C09144=1173.692,390.486,-82.941,-176.048,9.091,148.691
C09145=1173.688,390.734,-82.976,-176.048,9.094,148.691
C09146=1173.685,390.981,-83.012,-176.048,9.097,148.692
C09147=1173.681,391.228,-83.048,-176.047,9.099,148.693
C09148=1173.676,391.513,-83.089,-176.048,9.103,148.694
C09149=1173.671,391.797,-83.131,-176.047,9.107,148.694
C09150=1173.666,392.082,-83.172,-176.047,9.109,148.695
C09151=1173.663,392.366,-83.213,-176.047,9.112,148.696
C09152=1173.658,392.614,-83.249,-176.047,9.115,148.697
C09153=1173.654,392.861,-83.285,-176.047,9.118,148.697
C09154=1173.651,393.109,-83.320,-176.047,9.121,148.698
C09155=1173.647,393.356,-83.356,-176.047,9.124,148.699
C09156=1173.643,393.604,-83.392,-176.047,9.126,148.699
C09157=1173.639,393.851,-83.428,-176.047,9.129,148.700
C09158=1173.636,394.099,-83.464,-176.046,9.132,148.701
C09159=1173.631,394.346,-83.499,-176.047,9.134,148.701
C09160=1173.627,394.593,-83.535,-176.047,9.137,148.702
C09161=1173.623,394.841,-83.570,-176.047,9.140,148.703
C09162=1173.619,395.088,-83.607,-176.047,9.142,148.704
C09163=1173.616,395.335,-83.643,-176.047,9.145,148.704
C09164=1173.611,395.583,-83.679,-176.047,9.147,148.705
C09165=1173.608,395.831,-83.715,-176.047,9.150,148.706
C09166=1173.604,396.078,-83.751,-176.047,9.152,148.706
C09167=1173.599,396.325,-83.787,-176.047,9.155,148.707
C09168=1173.596,396.572,-83.822,-176.048,9.157,148.708
C09169=1173.592,396.820,-83.858,-176.048,9.160,148.708
C09170=1173.588,397.067,-83.895,-176.048,9.162,148.709
C09171=1173.584,397.314,-83.930,-176.048,9.165,148.710
C09172=1173.580,397.562,-83.966,-176.048,9.167,148.711
C09173=1173.576,397.810,-84.002,-176.048,9.170,148.711
C09174=1173.573,398.057,-84.038,-176.048,9.172,148.712
C09175=1173.568,398.304,-84.074,-176.048,9.175,148.713
C09176=1173.564,398.551,-84.109,-176.048,9.177,148.713
C09177=1173.561,398.798,-84.146,-176.049,9.180,148.714
C09178=1173.556,399.046,-84.182,-176.049,9.183,148.715
C09179=1173.553,399.293,-84.217,-176.049,9.185,148.715
C09180=1173.548,399.541,-84.253,-176.049,9.187,148.716
C09181=1173.545,399.788,-84.290,-176.049,9.189,148.717
C09182=1173.541,400.036,-84.325,-176.049,9.192,148.717
C09183=1173.537,400.283,-84.361,-176.050,9.194,148.718
C09184=1173.533,400.530,-84.398,-176.050,9.197,148.719
C09185=1173.529,400.778,-84.434,-176.050,9.198,148.719
C09186=1173.525,401.026,-84.469,-176.050,9.201,148.720
C09187=1173.521,401.272,-84.505,-176.050,9.203,148.721
C09188=1173.517,401.520,-84.541,-176.050,9.206,148.721
C09189=1173.513,401.767,-84.577,-176.051,9.208,148.722
C09190=1173.509,402.014,-84.614,-176.051,9.210,148.722
C09191=1173.506,402.262,-84.649,-176.051,9.213,148.723
C09192=1173.501,402.510,-84.686,-176.052,9.214,148.724
C09193=1173.498,402.757,-84.722,-176.052,9.217,148.725
C09194=1173.494,403.004,-84.757,-176.052,9.219,148.725
C09195=1173.490,403.252,-84.793,-176.052,9.221,148.726
C09196=1173.486,403.499,-84.830,-176.053,9.223,148.726
C09197=1173.482,403.747,-84.866,-176.052,9.226,148.727
C09198=1173.479,403.993,-84.902,-176.053,9.227,148.728
C09199=1173.474,404.240,-84.938,-176.053,9.230,148.728
C09200=1173.470,404.488,-84.973,-176.053,9.233,148.729
C09201=1173.467,404.735,-85.010,-176.054,9.234,148.729
C09202=1173.462,404.983,-85.046,-176.054,9.237,148.730
C09203=1173.459,405.230,-85.081,-176.054,9.238,148.731
C09204=1173.455,405.477,-85.118,-176.054,9.241,148.731
C09205=1173.451,405.725,-85.154,-176.055,9.242,148.732
C09206=1173.447,405.972,-85.191,-176.055,9.245,148.733
C09207=1173.443,406.220,-85.226,-176.055,9.246,148.733
C09208=1173.439,406.467,-85.262,-176.056,9.249,148.734
C09209=1173.435,406.714,-85.299,-176.055,9.251,148.734
C09210=1173.432,406.962,-85.334,-176.056,9.253,148.735
C09211=1173.428,407.209,-85.371,-176.056,9.255,148.736
C09212=1173.424,407.456,-85.407,-176.056,9.257,148.736
C09213=1173.420,407.704,-85.443,-176.057,9.259,148.737
C09214=1173.416,407.951,-85.479,-176.057,9.261,148.737
C09215=1173.412,408.199,-85.515,-176.057,9.263,148.738
C09216=1173.408,408.445,-85.551,-176.058,9.265,148.739
C09217=1173.403,408.693,-85.587,-176.058,9.267,148.739
C09218=1173.400,408.940,-85.623,-176.058,9.269,148.740
C09219=1173.396,409.188,-85.660,-176.058,9.271,148.740
C09220=1173.392,409.435,-85.695,-176.059,9.273,148.741
C09221=1173.388,409.682,-85.732,-176.059,9.275,148.742
C09222=1173.384,409.930,-85.768,-176.059,9.277,148.742
C09223=1173.381,410.177,-85.804,-176.059,9.279,148.743
C09224=1173.376,410.425,-85.840,-176.059,9.281,148.743
C09225=1173.373,410.672,-85.875,-176.060,9.283,148.744
C09226=1173.369,410.919,-85.912,-176.060,9.284,148.745
C09227=1173.365,411.167,-85.948,-176.060,9.287,148.745
C09228=1173.361,411.414,-85.985,-176.061,9.288,148.746
C09229=1173.357,411.661,-86.020,-176.061,9.291,148.746
C09230=1173.353,411.909,-86.057,-176.061,9.292,148.747
C09231=1173.350,412.156,-86.093,-176.062,9.294,148.747
C09232=1173.345,412.403,-86.130,-176.061,9.296,148.748
C09233=1173.342,412.651,-86.165,-176.062,9.298,148.749
C09234=1173.338,412.898,-86.202,-176.062,9.300,148.749
C09235=1173.334,413.145,-86.238,-176.062,9.302,148.750
C09236=1173.330,413.393,-86.274,-176.063,9.303,148.750
C09237=1173.326,413.640,-86.310,-176.063,9.306,148.751
C09238=1173.322,413.887,-86.347,-176.063,9.307,148.751
C09239=1173.318,414.135,-86.382,-176.064,9.309,148.752
C09240=1173.314,414.383,-86.418,-176.063,9.311,148.752
C09241=1173.310,414.629,-86.454,-176.064,9.313,148.753
C09242=1173.306,414.877,-86.491,-176.064,9.314,148.753
C09243=1173.302,415.124,-86.527,-176.064,9.316,148.754
C09244=1173.298,415.371,-86.563,-176.065,9.318,148.755
C09245=1173.295,415.619,-86.600,-176.065,9.320,148.755
C09246=1173.292,415.866,-86.636,-176.065,9.322,148.756
C09247=1173.291,416.113,-86.672,-176.065,9.323,148.756
C09248=1173.290,416.376,-86.709,-176.065,9.325,148.756
C09249=1173.291,416.639,-86.748,-176.065,9.327,148.757
C09250=1173.293,416.901,-86.785,-176.066,9.329,148.758
C09251=1173.296,417.163,-86.823,-176.066,9.330,148.758
C09252=1172.876,417.164,-86.867,-176.069,9.341,148.762
C09253=1172.873,416.899,-86.829,-176.069,9.339,148.761
C09254=1172.871,416.634,-86.790,-176.068,9.338,148.761
C09255=1172.869,416.368,-86.752,-176.069,9.336,148.760
C09256=1172.870,416.102,-86.714,-176.068,9.334,148.760
C09257=1172.872,415.855,-86.678,-176.068,9.333,148.759
C09258=1172.874,415.607,-86.642,-176.068,9.330,148.759
C09259=1172.877,415.361,-86.606,-176.068,9.329,148.758
C09260=1172.882,415.113,-86.570,-176.067,9.327,148.758
C09261=1172.885,414.866,-86.533,-176.067,9.325,148.757
C09262=1172.889,414.618,-86.497,-176.067,9.323,148.757
C09263=1172.893,414.371,-86.461,-176.067,9.322,148.756
C09264=1172.897,414.123,-86.425,-176.066,9.319,148.755
C09265=1172.901,413.876,-86.389,-176.066,9.318,148.755
C09266=1172.905,413.629,-86.352,-176.066,9.317,148.754
C09267=1172.908,413.382,-86.316,-176.066,9.314,148.754
C09268=1172.913,413.134,-86.280,-176.065,9.313,148.753
C09269=1172.916,412.887,-86.244,-176.065,9.311,148.753
C09270=1172.921,412.639,-86.208,-176.065,9.309,148.752
C09271=1172.924,412.392,-86.171,-176.065,9.307,148.752
C09272=1172.928,412.145,-86.135,-176.065,9.305,148.751
C09273=1172.932,411.898,-86.099,-176.064,9.303,148.751
C09274=1172.936,411.650,-86.063,-176.064,9.301,148.750
C09275=1172.939,411.403,-86.026,-176.064,9.299,148.749
C09276=1172.944,411.155,-85.990,-176.063,9.297,148.749
C09277=1172.947,410.908,-85.954,-176.063,9.296,148.748
C09278=1172.952,410.661,-85.918,-176.063,9.293,148.748
C09279=1172.955,410.413,-85.882,-176.062,9.292,148.747
C09280=1172.959,410.166,-85.846,-176.062,9.289,148.746
C09281=1172.963,409.918,-85.810,-176.062,9.288,148.746
C09282=1172.967,409.671,-85.773,-176.062,9.285,148.745
C09283=1172.971,409.424,-85.738,-176.061,9.284,148.745
C09284=1172.975,409.176,-85.701,-176.061,9.282,148.744
C09285=1172.978,408.929,-85.665,-176.061,9.280,148.744
C09286=1172.983,408.682,-85.629,-176.060,9.278,148.743
C09287=1172.987,408.435,-85.593,-176.061,9.276,148.742
C09288=1172.991,408.187,-85.557,-176.060,9.274,148.742
C09289=1172.995,407.940,-85.521,-176.060,9.272,148.741
C09290=1172.999,407.692,-85.485,-176.059,9.270,148.741
C09291=1173.002,407.446,-85.448,-176.059,9.268,148.740
C09292=1173.006,407.198,-85.413,-176.059,9.266,148.739
C09293=1173.010,406.951,-85.376,-176.059,9.264,148.739
C09294=1173.014,406.703,-85.340,-176.059,9.262,148.738
C09295=1173.018,406.456,-85.304,-176.058,9.260,148.738
C09296=1173.022,406.209,-85.268,-176.058,9.258,148.737
C09297=1173.026,405.961,-85.232,-176.058,9.256,148.736
C09298=1173.029,405.714,-85.196,-176.057,9.254,148.736
C09299=1173.034,405.466,-85.159,-176.057,9.251,148.735
C09300=1173.037,405.219,-85.124,-176.057,9.250,148.735
C09301=1173.041,404.971,-85.087,-176.057,9.247,148.734
C09302=1173.045,404.724,-85.051,-176.056,9.246,148.733
C09303=1173.048,404.477,-85.015,-176.056,9.243,148.733
C09304=1173.053,404.230,-84.979,-176.056,9.241,148.732
C09305=1173.057,403.983,-84.944,-176.055,9.239,148.731
C09306=1173.061,403.735,-84.907,-176.055,9.236,148.731
C09307=1173.065,403.488,-84.871,-176.055,9.235,148.730
C09308=1173.069,403.240,-84.835,-176.055,9.232,148.729
C09309=1173.073,402.993,-84.799,-176.055,9.230,148.729
C09310=1173.077,402.745,-84.763,-176.054,9.228,148.728
C09311=1173.081,402.498,-84.727,-176.054,9.226,148.727
C09312=1173.084,402.251,-84.691,-176.054,9.223,148.727
C09313=1173.088,402.003,-84.655,-176.053,9.221,148.726
C09314=1173.092,401.756,-84.619,-176.053,9.219,148.725
C09315=1173.096,401.508,-84.583,-176.053,9.217,148.725
C09316=1173.100,401.261,-84.547,-176.053,9.214,148.724
C09317=1173.103,401.014,-84.511,-176.053,9.212,148.724
C09318=1173.108,400.767,-84.475,-176.052,9.210,148.723
C09319=1173.112,400.519,-84.439,-176.052,9.207,148.722
C09320=1173.116,400.272,-84.403,-176.052,9.205,148.721
C09321=1173.120,400.025,-84.367,-176.052,9.203,148.721
C09322=1173.124,399.777,-84.331,-176.052,9.201,148.720
C09323=1173.127,399.530,-84.295,-176.051,9.198,148.719
C09324=1173.131,399.283,-84.259,-176.051,9.195,148.719
C09325=1173.135,399.035,-84.223,-176.051,9.193,148.718
C09326=1173.139,398.787,-84.187,-176.050,9.191,148.717
C09327=1173.143,398.540,-84.151,-176.051,9.189,148.717
C09328=1173.147,398.293,-84.115,-176.051,9.186,148.716
C09329=1173.151,398.046,-84.080,-176.050,9.184,148.715
C09330=1173.155,397.799,-84.043,-176.050,9.181,148.715
C09331=1173.159,397.551,-84.007,-176.050,9.179,148.714
C09332=1173.163,397.303,-83.971,-176.050,9.176,148.713
C09333=1173.167,397.056,-83.936,-176.050,9.174,148.713
C09334=1173.170,396.809,-83.899,-176.050,9.171,148.712
C09335=1173.175,396.561,-83.863,-176.050,9.169,148.711
C09336=1173.178,396.314,-83.828,-176.050,9.166,148.711
C09337=1173.182,396.067,-83.791,-176.050,9.164,148.710
C09338=1173.187,395.820,-83.756,-176.049,9.161,148.709
C09339=1173.190,395.572,-83.720,-176.049,9.158,148.708
C09340=1173.195,395.324,-83.684,-176.049,9.156,148.708
C09341=1173.198,395.077,-83.648,-176.049,9.153,148.707
C09342=1173.202,394.830,-83.612,-176.049,9.151,148.706
C09343=1173.206,394.582,-83.576,-176.049,9.148,148.706
C09344=1173.210,394.335,-83.541,-176.049,9.146,148.705
C09345=1173.214,394.087,-83.505,-176.049,9.142,148.704
C09346=1173.218,393.840,-83.468,-176.049,9.140,148.704
C09347=1173.222,393.593,-83.433,-176.049,9.137,148.703
C09348=1173.226,393.346,-83.397,-176.049,9.135,148.702
C09349=1173.230,393.098,-83.361,-176.049,9.132,148.701
C09350=1173.233,392.851,-83.325,-176.049,9.129,148.701
C09351=1173.237,392.603,-83.289,-176.049,9.126,148.700
C09352=1173.241,392.356,-83.253,-176.049,9.124,148.699
C09353=1173.246,392.071,-83.213,-176.049,9.120,148.698
C09354=1173.250,391.786,-83.171,-176.049,9.118,148.698
C09355=1173.255,391.501,-83.130,-176.049,9.114,148.697
C09356=1173.259,391.217,-83.089,-176.049,9.111,148.696
C09357=1173.263,390.970,-83.053,-176.050,9.108,148.696
C09358=1173.267,390.722,-83.017,-176.050,9.105,148.695
C09359=1173.271,390.475,-82.982,-176.050,9.102,148.694
C09360=1173.276,390.227,-82.946,-176.050,9.099,148.693
C09361=1173.279,389.981,-82.910,-176.050,9.096,148.693
C09362=1173.283,389.733,-82.874,-176.051,9.093,148.692
C09363=1173.286,389.486,-82.839,-176.051,9.091,148.691
C09364=1173.291,389.238,-82.802,-176.051,9.087,148.690
C09365=1173.295,388.991,-82.767,-176.051,9.085,148.690
C09366=1173.299,388.743,-82.732,-176.052,9.081,148.689
C09367=1173.302,388.496,-82.696,-176.052,9.078,148.688
C09368=1173.307,388.248,-82.660,-176.052,9.076,148.688
C09369=1173.310,388.001,-82.624,-176.053,9.072,148.687
C09370=1173.314,387.754,-82.588,-176.052,9.070,148.686
C09371=1173.319,387.507,-82.552,-176.053,9.067,148.686
C09372=1173.322,387.259,-82.517,-176.054,9.063,148.685
C09373=1173.326,387.012,-82.481,-176.054,9.060,148.684
C09374=1173.330,386.764,-82.446,-176.054,9.058,148.684
C09375=1173.333,386.517,-82.410,-176.055,9.054,148.683
C09376=1173.338,386.269,-82.374,-176.055,9.051,148.682
C09377=1173.342,386.022,-82.339,-176.056,9.048,148.681
C09378=1173.346,385.775,-82.303,-176.056,9.044,148.681
C09379=1173.349,385.527,-82.268,-176.057,9.041,148.680
C09380=1173.354,385.279,-82.232,-176.058,9.038,148.679
C09381=1173.357,385.032,-82.196,-176.058,9.035,148.679
C09382=1173.362,384.785,-82.161,-176.059,9.031,148.678
C09383=1173.365,384.537,-82.125,-176.059,9.028,148.677
C09384=1173.369,384.290,-82.090,-176.060,9.025,148.677
C09385=1173.373,384.042,-82.054,-176.061,9.022,148.676
C09386=1173.377,383.795,-82.018,-176.061,9.018,148.675
C09387=1173.381,383.548,-81.983,-176.062,9.015,148.674
C09388=1173.385,383.300,-81.947,-176.063,9.012,148.674
C09389=1173.389,383.053,-81.912,-176.064,9.009,148.673
C09390=1173.392,382.805,-81.876,-176.064,9.006,148.673
C09391=1173.398,382.558,-81.841,-176.065,9.002,148.672
C09392=1173.401,382.310,-81.806,-176.066,8.998,148.671
C09393=1173.405,382.063,-81.770,-176.067,8.995,148.671
C09394=1173.409,381.815,-81.735,-176.067,8.992,148.670
C09395=1173.413,381.568,-81.699,-176.068,8.989,148.669
C09396=1173.416,381.321,-81.664,-176.069,8.986,148.669
C09397=1173.420,381.073,-81.628,-176.070,8.982,148.668
C09398=1173.425,380.825,-81.592,-176.071,8.979,148.667
C09399=1173.429,380.578,-81.558,-176.071,8.975,148.667
C09400=1173.433,380.331,-81.522,-176.073,8.971,148.666
C09401=1173.436,380.083,-81.487,-176.074,8.968,148.665
C09402=1173.440,379.836,-81.451,-176.074,8.965,148.665
C09403=1173.444,379.589,-81.416,-176.076,8.961,148.664
C09404=1173.448,379.341,-81.380,-176.077,8.958,148.664
C09405=1173.452,379.093,-81.345,-176.078,8.954,148.663
C09406=1173.456,378.846,-81.310,-176.079,8.951,148.662
C09407=1173.460,378.599,-81.275,-176.080,8.947,148.662
C09408=1173.464,378.351,-81.239,-176.081,8.944,148.661
C09409=1173.468,378.103,-81.204,-176.082,8.940,148.660
C09410=1173.473,377.856,-81.169,-176.083,8.937,148.660
C09411=1173.476,377.609,-81.133,-176.084,8.933,148.659
C09412=1173.480,377.361,-81.098,-176.086,8.930,148.659
C09413=1173.484,377.114,-81.063,-176.087,8.926,148.658
C09414=1173.488,376.866,-81.028,-176.088,8.923,148.658
C09415=1173.492,376.619,-80.992,-176.089,8.919,148.657
C09416=1173.496,376.371,-80.957,-176.091,8.915,148.656
C09417=1173.500,376.124,-80.922,-176.092,8.912,148.656
C09418=1173.504,375.876,-80.886,-176.093,8.908,148.655
C09419=1173.508,375.628,-80.852,-176.095,8.905,148.655
C09420=1173.512,375.381,-80.816,-176.096,8.902,148.654
C09421=1173.516,375.134,-80.781,-176.097,8.898,148.653
C09422=1173.519,374.886,-80.746,-176.098,8.894,148.653
C09423=1173.524,374.639,-80.711,-176.100,8.891,148.652
C09424=1173.527,374.391,-80.675,-176.101,8.887,148.652
C09425=1173.531,374.144,-80.641,-176.103,8.883,148.651
C09426=1173.535,373.897,-80.606,-176.104,8.879,148.651
C09427=1173.539,373.649,-80.571,-176.105,8.876,148.650
C09428=1173.543,373.402,-80.536,-176.107,8.872,148.650
C09429=1173.547,373.154,-80.501,-176.108,8.869,148.649
C09430=1173.551,372.906,-80.465,-176.110,8.865,148.649
C09431=1173.555,372.659,-80.431,-176.112,8.861,148.648
C09432=1173.559,372.411,-80.395,-176.113,8.857,148.647
C09433=1173.563,372.163,-80.361,-176.114,8.855,148.647
C09434=1173.567,371.916,-80.325,-176.116,8.851,148.646
C09435=1173.571,371.668,-80.291,-176.118,8.847,148.646
C09436=1173.575,371.422,-80.256,-176.119,8.843,148.646
C09437=1173.579,371.174,-80.221,-176.121,8.840,148.645
C09438=1173.582,370.926,-80.186,-176.123,8.836,148.645
C09439=1173.587,370.679,-80.151,-176.125,8.832,148.644
C09440=1173.591,370.431,-80.116,-176.126,8.828,148.643
C09441=1173.595,370.184,-80.081,-176.128,8.825,148.643
C09442=1173.599,369.936,-80.046,-176.130,8.821,148.643
C09443=1173.603,369.689,-80.012,-176.131,8.817,148.642
C09444=1173.607,369.441,-79.977,-176.133,8.814,148.642
C09445=1173.611,369.193,-79.942,-176.135,8.810,148.641
C09446=1173.615,368.946,-79.907,-176.137,8.806,148.641
C09447=1173.619,368.698,-79.872,-176.138,8.803,148.640
C09448=1173.623,368.451,-79.838,-176.140,8.799,148.640
C09449=1173.626,368.203,-79.803,-176.142,8.795,148.639
C09450=1173.631,367.956,-79.768,-176.143,8.792,148.639
C09451=1173.635,367.708,-79.733,-176.145,8.788,148.638
C09452=1173.638,367.461,-79.699,-176.147,8.785,148.638
C09453=1173.642,367.213,-79.664,-176.149,8.781,148.637
C09454=1173.647,366.966,-79.629,-176.151,8.777,148.637
C09455=1173.651,366.718,-79.595,-176.153,8.774,148.637
C09456=1173.655,366.471,-79.561,-176.154,8.770,148.636
C09457=1173.659,366.188,-79.521,-176.157,8.766,148.636
C09458=1173.664,365.907,-79.481,-176.159,8.762,148.635
C09459=1173.668,365.624,-79.442,-176.161,8.758,148.635
C09460=1173.673,365.343,-79.402,-176.164,8.753,148.634
C09461=1173.676,365.095,-79.368,-176.165,8.750,148.634
C09462=1173.681,364.847,-79.333,-176.167,8.746,148.633
C09463=1173.685,364.599,-79.299,-176.169,8.743,148.633
C09464=1173.688,364.353,-79.264,-176.171,8.739,148.633
C09465=1173.692,364.105,-79.229,-176.174,8.735,148.632
C09466=1173.697,363.857,-79.195,-176.176,8.731,148.632
C09467=1173.701,363.610,-79.161,-176.178,8.728,148.632
C09468=1173.705,363.362,-79.126,-176.180,8.724,148.631
C09469=1173.709,363.115,-79.092,-176.182,8.720,148.631
C09470=1173.712,362.867,-79.057,-176.184,8.717,148.631
C09471=1173.717,362.619,-79.023,-176.186,8.713,148.630
C09472=1173.720,362.372,-78.989,-176.188,8.709,148.630
C09473=1173.725,362.124,-78.954,-176.190,8.706,148.629
C09474=1173.728,361.876,-78.920,-176.192,8.702,148.629
C09475=1173.733,361.629,-78.885,-176.194,8.699,148.629
C09476=1173.736,361.382,-78.852,-176.197,8.694,148.628
C09477=1173.740,361.134,-78.817,-176.199,8.691,148.628
C09478=1173.745,360.886,-78.782,-176.201,8.688,148.628
C09479=1173.748,360.639,-78.748,-176.203,8.684,148.627
C09480=1173.753,360.391,-78.714,-176.205,8.681,148.627
C09481=1173.757,360.143,-78.680,-176.207,8.676,148.627
C09482=1173.761,359.895,-78.646,-176.210,8.673,148.626
C09483=1173.765,359.648,-78.612,-176.212,8.669,148.626
C09484=1173.769,359.400,-78.577,-176.214,8.666,148.626
C09485=1173.773,359.153,-78.543,-176.216,8.662,148.625
C09486=1173.777,358.905,-78.509,-176.219,8.658,148.625
C09487=1173.781,358.657,-78.475,-176.221,8.655,148.625
C09488=1173.785,358.410,-78.441,-176.223,8.651,148.624
C09489=1173.789,358.163,-78.407,-176.225,8.648,148.624
C09490=1173.792,357.915,-78.372,-176.227,8.644,148.624
C09491=1173.797,357.667,-78.338,-176.230,8.640,148.623
C09492=1173.801,357.420,-78.305,-176.232,8.637,148.623
C09493=1173.805,357.171,-78.270,-176.234,8.633,148.623
C09494=1173.809,356.924,-78.236,-176.236,8.630,148.623
C09495=1173.813,356.677,-78.203,-176.239,8.626,148.622
C09496=1173.817,356.428,-78.168,-176.241,8.622,148.622
C09497=1173.821,356.181,-78.134,-176.243,8.619,148.622
C09498=1173.826,355.933,-78.101,-176.245,8.616,148.621
C09499=1173.829,355.686,-78.066,-176.248,8.611,148.621
C09500=1173.833,355.438,-78.032,-176.250,8.608,148.621
C09501=1173.838,355.190,-77.999,-176.252,8.605,148.621
C09502=1173.841,354.943,-77.964,-176.255,8.601,148.620
C09503=1173.845,354.695,-77.931,-176.256,8.598,148.620
C09504=1173.850,354.447,-77.897,-176.259,8.594,148.620
C09505=1173.853,354.200,-77.863,-176.261,8.590,148.619
C09506=1173.857,353.952,-77.829,-176.264,8.587,148.619
C09507=1173.861,353.704,-77.795,-176.266,8.583,148.619
C09508=1173.866,353.457,-77.762,-176.268,8.580,148.619
C09509=1173.869,353.210,-77.728,-176.271,8.576,148.618
C09510=1173.873,352.961,-77.694,-176.273,8.573,148.618
C09511=1173.878,352.714,-77.660,-176.275,8.569,148.618
C09512=1173.882,352.466,-77.627,-176.277,8.566,148.617
C09513=1173.885,352.219,-77.593,-176.279,8.562,148.617
C09514=1173.889,351.970,-77.559,-176.282,8.558,148.617
C09515=1173.894,351.723,-77.525,-176.285,8.555,148.617
C09516=1173.898,351.475,-77.492,-176.287,8.552,148.616
C09517=1173.902,351.228,-77.459,-176.289,8.548,148.616
C09518=1173.906,350.981,-77.425,-176.291,8.545,148.616
C09519=1173.910,350.732,-77.391,-176.294,8.541,148.616
C09520=1173.914,350.484,-77.357,-176.296,8.537,148.615
C09521=1173.918,350.237,-77.324,-176.298,8.534,148.615
C09522=1173.922,349.989,-77.290,-176.301,8.531,148.615
C09523=1173.926,349.741,-77.257,-176.303,8.527,148.615
C09524=1173.930,349.494,-77.223,-176.306,8.523,148.614
C09525=1173.934,349.246,-77.189,-176.308,8.520,148.614
C09526=1173.938,348.998,-77.156,-176.310,8.516,148.614
C09527=1173.942,348.751,-77.122,-176.312,8.513,148.614
C09528=1173.946,348.503,-77.089,-176.314,8.510,148.613
C09529=1173.951,348.255,-77.056,-176.317,8.506,148.613
C09530=1173.955,348.008,-77.023,-176.319,8.502,148.613
C09531=1173.959,347.760,-76.989,-176.322,8.499,148.613
C09532=1173.963,347.512,-76.955,-176.324,8.496,148.612
C09533=1173.967,347.264,-76.922,-176.326,8.492,148.612
C09534=1173.971,347.016,-76.889,-176.329,8.489,148.612
C09535=1173.975,346.769,-76.855,-176.331,8.486,148.612
C09536=1173.979,346.521,-76.822,-176.334,8.482,148.612
C09537=1173.984,346.273,-76.789,-176.336,8.478,148.611
C09538=1173.987,346.026,-76.755,-176.338,8.475,148.611
C09539=1173.991,345.778,-76.722,-176.341,8.472,148.611
C09540=1173.996,345.531,-76.689,-176.343,8.468,148.611
C09541=1174.000,345.283,-76.656,-176.345,8.465,148.610
C09542=1174.003,345.034,-76.622,-176.347,8.462,148.610
C09543=1174.007,344.787,-76.589,-176.350,8.458,148.610
C09544=1174.012,344.539,-76.556,-176.352,8.454,148.610
C09545=1174.016,344.291,-76.523,-176.355,8.451,148.610
C09546=1174.020,344.043,-76.490,-176.357,8.448,148.609
C09547=1174.024,343.796,-76.456,-176.359,8.445,148.609
C09548=1174.028,343.548,-76.423,-176.362,8.441,148.609
C09549=1174.032,343.300,-76.390,-176.364,8.438,148.609
C09550=1174.036,343.053,-76.357,-176.367,8.434,148.608
C09551=1174.041,342.805,-76.324,-176.369,8.430,148.608
C09552=1174.045,342.557,-76.291,-176.371,8.427,148.608
C09553=1174.049,342.309,-76.257,-176.374,8.424,148.608
C09554=1174.053,342.062,-76.224,-176.376,8.421,148.608
C09555=1174.057,341.813,-76.192,-176.379,8.418,148.608
C09556=1174.061,341.566,-76.159,-176.381,8.414,148.607
C09557=1174.065,341.318,-76.126,-176.384,8.410,148.607
C09558=1174.069,341.070,-76.093,-176.386,8.407,148.607
C09559=1174.073,340.823,-76.060,-176.388,8.404,148.607
C09560=1174.077,340.575,-76.027,-176.391,8.400,148.606
C09561=1174.082,340.295,-75.989,-176.393,8.396,148.606
C09562=1174.087,340.016,-75.953,-176.396,8.393,148.606
C09563=1174.091,339.737,-75.916,-176.399,8.389,148.606
C09564=1174.097,339.458,-75.879,-176.402,8.385,148.606
C09565=1174.100,339.210,-75.846,-176.404,8.382,148.605
C09566=1174.104,338.963,-75.813,-176.406,8.378,148.605
C09567=1174.108,338.714,-75.780,-176.409,8.375,148.605
C09568=1174.113,338.466,-75.747,-176.411,8.372,148.605
C09569=1174.117,338.219,-75.714,-176.414,8.369,148.605
C09570=1174.120,337.971,-75.682,-176.416,8.365,148.605
C09571=1174.125,337.723,-75.649,-176.418,8.362,148.604
C09572=1174.129,337.475,-75.616,-176.420,8.359,148.604
C09573=1174.133,337.227,-75.584,-176.423,8.355,148.604
C09574=1174.137,336.979,-75.551,-176.426,8.352,148.604
C09575=1174.141,336.732,-75.518,-176.428,8.348,148.604
C09576=1174.146,336.484,-75.486,-176.431,8.345,148.604
C09577=1174.149,336.237,-75.453,-176.433,8.342,148.603
C09578=1174.154,335.988,-75.421,-176.435,8.338,148.603
C09579=1174.158,335.741,-75.388,-176.438,8.335,148.603
C09580=1174.161,335.493,-75.356,-176.440,8.332,148.603
C09581=1174.166,335.245,-75.323,-176.442,8.329,148.603
C09582=1174.170,334.996,-75.290,-176.445,8.325,148.603
C09583=1174.173,334.749,-75.258,-176.448,8.322,148.602
C09584=1174.178,334.501,-75.225,-176.450,8.318,148.602
C09585=1174.183,334.254,-75.192,-176.452,8.315,148.602
C09586=1174.186,334.006,-75.161,-176.455,8.312,148.602
C09587=1174.190,333.758,-75.127,-176.457,8.309,148.602
C09588=1174.195,333.510,-75.095,-176.460,8.305,148.602
C09589=1174.198,333.262,-75.062,-176.462,8.302,148.601
C09590=1174.203,333.014,-75.030,-176.464,8.299,148.601
C09591=1174.207,332.767,-74.998,-176.467,8.296,148.601
C09592=1174.211,332.519,-74.965,-176.469,8.293,148.601
C09593=1174.216,332.270,-74.933,-176.472,8.289,148.601
C09594=1174.219,332.023,-74.900,-176.475,8.285,148.601
C09595=1174.224,331.775,-74.868,-176.477,8.282,148.601
C09596=1174.228,331.527,-74.836,-176.479,8.279,148.600
C09597=1174.232,331.280,-74.803,-176.482,8.276,148.600
C09598=1174.236,331.032,-74.771,-176.484,8.273,148.600
C09599=1174.240,330.783,-74.739,-176.487,8.269,148.600
C09600=1174.244,330.535,-74.707,-176.489,8.266,148.600
C09601=1174.249,330.288,-74.674,-176.492,8.263,148.600
C09602=1174.252,330.040,-74.642,-176.494,8.260,148.600
C09603=1174.257,329.792,-74.610,-176.496,8.256,148.599
C09604=1174.260,329.544,-74.578,-176.499,8.253,148.599
C09605=1174.265,329.297,-74.545,-176.501,8.250,148.599
C09606=1174.269,329.049,-74.514,-176.504,8.247,148.599
C09607=1174.273,328.800,-74.481,-176.507,8.243,148.599
C09608=1174.277,328.552,-74.449,-176.509,8.240,148.599
C09609=1174.282,328.305,-74.417,-176.512,8.237,148.599
C09610=1174.286,328.057,-74.385,-176.514,8.233,148.598
C09611=1174.290,327.809,-74.352,-176.516,8.230,148.598
C09612=1174.294,327.561,-74.320,-176.519,8.227,148.598
C09613=1174.298,327.313,-74.289,-176.521,8.224,148.598
C09614=1174.302,327.065,-74.256,-176.524,8.220,148.598
C09615=1174.306,326.817,-74.225,-176.526,8.217,148.598
C09616=1174.310,326.570,-74.193,-176.529,8.214,148.598
C09617=1174.315,326.321,-74.161,-176.531,8.211,148.598
C09618=1174.319,326.073,-74.129,-176.534,8.208,148.597
C09619=1174.324,325.826,-74.097,-176.536,8.205,148.597
C09620=1174.327,325.578,-74.065,-176.539,8.202,148.597
C09621=1174.331,325.330,-74.033,-176.541,8.198,148.597
C09622=1174.335,325.081,-74.001,-176.544,8.195,148.597
C09623=1174.340,324.834,-73.969,-176.546,8.192,148.597
C09624=1174.343,324.586,-73.937,-176.549,8.189,148.597
C09625=1174.347,324.338,-73.905,-176.551,8.186,148.597
C09626=1174.352,324.090,-73.873,-176.554,8.182,148.596
C09627=1174.356,323.842,-73.842,-176.557,8.179,148.596
C09628=1174.360,323.595,-73.810,-176.559,8.175,148.596
C09629=1174.365,323.346,-73.778,-176.562,8.172,148.596
C09630=1174.369,323.098,-73.746,-176.564,8.169,148.596
C09631=1174.373,322.850,-73.715,-176.567,8.166,148.596
C09632=1174.377,322.602,-73.683,-176.569,8.163,148.596
C09633=1174.380,322.354,-73.651,-176.571,8.159,148.596
C09634=1174.385,322.107,-73.619,-176.574,8.156,148.596
C09635=1174.389,321.859,-73.587,-176.576,8.153,148.595
C09636=1174.394,321.611,-73.557,-176.579,8.150,148.595
C09637=1174.397,321.363,-73.525,-176.581,8.147,148.595
C09638=1174.401,321.115,-73.493,-176.584,8.144,148.595
C09639=1174.406,320.867,-73.461,-176.586,8.140,148.595
C09640=1174.410,320.618,-73.430,-176.589,8.137,148.595
C09641=1174.415,320.371,-73.398,-176.591,8.134,148.595
C09642=1174.418,320.123,-73.366,-176.594,8.131,148.595
C09643=1174.422,319.875,-73.335,-176.596,8.128,148.595
C09644=1174.427,319.627,-73.304,-176.599,8.125,148.595
C09645=1174.431,319.379,-73.271,-176.601,8.122,148.595
C09646=1174.435,319.131,-73.240,-176.604,8.119,148.595
C09647=1174.439,318.883,-73.209,-176.606,8.115,148.594
C09648=1174.444,318.635,-73.177,-176.609,8.112,148.594
C09649=1174.448,318.387,-73.146,-176.611,8.109,148.594
C09650=1174.452,318.139,-73.115,-176.614,8.106,148.594
C09651=1174.456,317.891,-73.083,-176.616,8.103,148.594
C09652=1174.460,317.643,-73.052,-176.619,8.100,148.594
C09653=1174.464,317.395,-73.020,-176.621,8.096,148.594
C09654=1174.469,317.147,-72.989,-176.624,8.093,148.594
C09655=1174.472,316.899,-72.958,-176.626,8.090,148.594
C09656=1174.477,316.651,-72.927,-176.629,8.087,148.594
C09657=1174.481,316.403,-72.895,-176.631,8.084,148.593
C09658=1174.485,316.155,-72.864,-176.634,8.081,148.593
C09659=1174.489,315.907,-72.832,-176.637,8.078,148.593
C09660=1174.494,315.659,-72.802,-176.639,8.075,148.593
C09661=1174.497,315.411,-72.770,-176.642,8.072,148.593
C09662=1174.502,315.163,-72.739,-176.644,8.068,148.593
C09663=1174.506,314.915,-72.707,-176.647,8.065,148.593
C09664=1174.510,314.667,-72.676,-176.649,8.062,148.593
C09665=1174.515,314.391,-72.641,-176.652,8.058,148.593
C09666=1174.520,314.114,-72.606,-176.655,8.055,148.593
C09667=1174.524,313.837,-72.572,-176.658,8.051,148.593
C09668=1174.529,313.560,-72.537,-176.660,8.048,148.593
C09669=1174.533,313.311,-72.506,-176.663,8.045,148.592
C09670=1174.537,313.064,-72.475,-176.665,8.042,148.592
C09671=1174.541,312.815,-72.444,-176.668,8.039,148.592
C09672=1174.546,312.567,-72.413,-176.670,8.036,148.592
C09673=1174.550,312.320,-72.381,-176.673,8.033,148.592
C09674=1174.554,312.071,-72.350,-176.675,8.029,148.592
C09675=1174.559,311.823,-72.319,-176.678,8.026,148.592
C09676=1174.563,311.575,-72.288,-176.681,8.023,148.592
C09677=1174.567,311.327,-72.257,-176.683,8.020,148.592
C09678=1174.571,311.080,-72.226,-176.686,8.017,148.592
C09679=1174.575,310.831,-72.196,-176.688,8.014,148.592
C09680=1174.579,310.583,-72.165,-176.691,8.011,148.592
C09681=1174.584,310.335,-72.134,-176.694,8.008,148.592
C09682=1174.588,310.087,-72.102,-176.696,8.004,148.592
C09683=1174.592,309.839,-72.071,-176.699,8.001,148.592
C09684=1174.596,309.592,-72.041,-176.701,7.998,148.591
C09685=1174.600,309.343,-72.010,-176.704,7.995,148.591
C09686=1174.605,309.095,-71.979,-176.706,7.992,148.591
C09687=1174.609,308.847,-71.949,-176.709,7.989,148.591
C09688=1174.613,308.598,-71.917,-176.711,7.986,148.591
C09689=1174.617,308.351,-71.887,-176.714,7.983,148.591
C09690=1174.622,308.103,-71.857,-176.716,7.980,148.591
C09691=1174.626,307.854,-71.825,-176.719,7.977,148.591
C09692=1174.631,307.606,-71.795,-176.722,7.974,148.591
C09693=1174.634,307.359,-71.764,-176.724,7.970,148.591
C09694=1174.638,307.110,-71.733,-176.726,7.968,148.591
C09695=1174.643,306.862,-71.703,-176.729,7.965,148.591
C09696=1174.647,306.614,-71.672,-176.731,7.962,148.591
C09697=1174.652,306.366,-71.642,-176.734,7.959,148.591
C09698=1174.656,306.118,-71.610,-176.736,7.956,148.591
C09699=1174.659,305.870,-71.580,-176.739,7.953,148.591
C09700=1174.664,305.622,-71.550,-176.742,7.950,148.591
C09701=1174.669,305.374,-71.519,-176.744,7.946,148.591
C09702=1174.672,305.126,-71.488,-176.747,7.943,148.591
C09703=1174.677,304.878,-71.457,-176.750,7.940,148.591
C09704=1174.681,304.630,-71.427,-176.752,7.937,148.590
C09705=1174.685,304.382,-71.397,-176.755,7.934,148.590
C09706=1174.689,304.133,-71.366,-176.757,7.931,148.590
C09707=1174.694,303.885,-71.335,-176.760,7.928,148.590
C09708=1174.698,303.637,-71.305,-176.762,7.925,148.590
C09709=1174.702,303.389,-71.274,-176.765,7.922,148.590
C09710=1174.706,303.141,-71.244,-176.768,7.919,148.590
C09711=1174.710,302.893,-71.213,-176.770,7.915,148.590
C09712=1174.715,302.644,-71.183,-176.773,7.913,148.590
C09713=1174.719,302.397,-71.153,-176.775,7.910,148.590
C09714=1174.724,302.149,-71.122,-176.777,7.907,148.590
C09715=1174.727,301.900,-71.092,-176.780,7.904,148.590
C09716=1174.732,301.652,-71.062,-176.783,7.901,148.590
C09717=1174.736,301.404,-71.031,-176.785,7.898,148.590
C09718=1174.740,301.156,-71.001,-176.788,7.895,148.590
C09719=1174.745,300.908,-70.971,-176.790,7.892,148.590
C09720=1174.749,300.660,-70.940,-176.793,7.889,148.590
C09721=1174.752,300.412,-70.910,-176.795,7.886,148.590
C09722=1174.757,300.163,-70.880,-176.798,7.883,148.590
C09723=1174.761,299.916,-70.850,-176.801,7.880,148.590
C09724=1174.766,299.667,-70.820,-176.804,7.877,148.590
C09725=1174.770,299.419,-70.789,-176.806,7.873,148.590
C09726=1174.775,299.171,-70.759,-176.809,7.870,148.590
C09727=1174.779,298.923,-70.729,-176.811,7.867,148.590
C09728=1174.782,298.675,-70.699,-176.813,7.865,148.590
C09729=1174.787,298.426,-70.669,-176.816,7.862,148.590
C09730=1174.791,298.178,-70.638,-176.818,7.859,148.590
C09731=1174.796,297.930,-70.608,-176.821,7.856,148.590
C09732=1174.800,297.682,-70.578,-176.824,7.853,148.590
C09733=1174.804,297.434,-70.549,-176.826,7.850,148.589
C09734=1174.809,297.186,-70.518,-176.829,7.847,148.590
C09735=1174.813,296.938,-70.489,-176.832,7.844,148.590
C09736=1174.817,296.690,-70.458,-176.834,7.841,148.590
C09737=1174.821,296.442,-70.428,-176.837,7.837,148.589
C09738=1174.825,296.194,-70.398,-176.839,7.834,148.589
C09739=1174.830,295.945,-70.368,-176.842,7.832,148.589
C09740=1174.834,295.696,-70.338,-176.844,7.829,148.590
C09741=1174.838,295.449,-70.308,-176.847,7.826,148.589
C09742=1174.842,295.200,-70.279,-176.849,7.823,148.589
C09743=1174.847,294.952,-70.248,-176.852,7.820,148.589
C09744=1174.851,294.704,-70.219,-176.855,7.817,148.589
C09745=1174.855,294.456,-70.189,-176.858,7.814,148.589
C09746=1174.860,294.208,-70.158,-176.860,7.811,148.589
C09747=1174.864,293.960,-70.129,-176.863,7.808,148.589
C09748=1174.868,293.711,-70.099,-176.865,7.805,148.589
C09749=1174.872,293.463,-70.070,-176.867,7.803,148.589
C09750=1174.877,293.215,-70.039,-176.870,7.800,148.589
C09751=1174.881,292.967,-70.010,-176.872,7.796,148.589
C09752=1174.885,292.719,-69.980,-176.875,7.793,148.589
C09753=1174.889,292.470,-69.951,-176.878,7.790,148.589
C09754=1174.893,292.223,-69.921,-176.881,7.787,148.589
C09755=1174.898,291.974,-69.891,-176.883,7.784,148.589
C09756=1174.902,291.726,-69.861,-176.886,7.781,148.589
C09757=1174.906,291.478,-69.832,-176.888,7.778,148.589
C09758=1174.911,291.229,-69.802,-176.891,7.776,148.589
C09759=1174.914,290.982,-69.772,-176.893,7.773,148.589
C09760=1174.919,290.733,-69.743,-176.896,7.770,148.589
C09761=1174.924,290.485,-69.713,-176.899,7.767,148.589
C09762=1174.928,290.237,-69.683,-176.901,7.764,148.589
C09763=1174.932,289.988,-69.654,-176.904,7.761,148.589
C09764=1174.936,289.740,-69.624,-176.907,7.758,148.589
C09765=1174.940,289.492,-69.595,-176.909,7.755,148.589
C09766=1174.944,289.244,-69.565,-176.911,7.753,148.589
C09767=1174.949,288.996,-69.536,-176.914,7.750,148.589
C09768=1174.953,288.748,-69.507,-176.916,7.746,148.589
C09769=1174.958,288.473,-69.473,-176.919,7.743,148.589
C09770=1174.963,288.198,-69.441,-176.922,7.740,148.589
C09771=1174.967,287.924,-69.408,-176.925,7.737,148.589
C09772=1174.972,287.648,-69.376,-176.928,7.734,148.589
C09773=1174.977,287.400,-69.346,-176.931,7.731,148.589
C09774=1174.981,287.152,-69.317,-176.933,7.728,148.589
C09775=1174.985,286.904,-69.288,-176.936,7.725,148.589
C09776=1174.989,286.655,-69.258,-176.939,7.722,148.589
C09777=1174.993,286.407,-69.229,-176.941,7.718,148.589
C09778=1174.998,286.160,-69.200,-176.943,7.716,148.589
C09779=1175.002,285.911,-69.170,-176.946,7.713,148.589
C09780=1175.007,285.662,-69.141,-176.949,7.710,148.589
C09781=1175.011,285.414,-69.112,-176.952,7.707,148.589
C09782=1175.015,285.166,-69.082,-176.954,7.704,148.589
C09783=1175.019,284.918,-69.053,-176.957,7.701,148.590
C09784=1175.024,284.670,-69.024,-176.959,7.699,148.590
C09785=1175.028,284.422,-68.994,-176.962,7.696,148.590
C09786=1175.033,284.173,-68.966,-176.964,7.693,148.589
C09787=1175.037,283.925,-68.936,-176.967,7.690,148.589
C09788=1175.041,283.676,-68.907,-176.970,7.687,148.590
C09789=1175.045,283.428,-68.877,-176.972,7.684,148.590
C09790=1175.050,283.180,-68.849,-176.975,7.681,148.590
C09791=1175.054,282.932,-68.820,-176.977,7.679,148.590
C09792=1175.058,282.684,-68.791,-176.980,7.676,148.590
C09793=1175.063,282.435,-68.762,-176.983,7.673,148.590
C09794=1175.067,282.187,-68.733,-176.986,7.670,148.590
C09795=1175.071,281.939,-68.703,-176.988,7.667,148.590
C09796=1175.076,281.690,-68.675,-176.991,7.664,148.590
C09797=1175.080,281.442,-68.645,-176.993,7.661,148.590
C09798=1175.084,281.194,-68.616,-176.995,7.658,148.590
C09799=1175.089,280.946,-68.588,-176.998,7.655,148.590
C09800=1175.093,280.697,-68.559,-177.001,7.653,148.590
C09801=1175.097,280.449,-68.529,-177.004,7.650,148.590
C09802=1175.102,280.200,-68.500,-177.006,7.647,148.590
C09803=1175.106,279.953,-68.472,-177.009,7.644,148.590
C09804=1175.110,279.704,-68.443,-177.011,7.641,148.590
C09805=1175.114,279.456,-68.414,-177.014,7.638,148.590
C09806=1175.119,279.208,-68.385,-177.017,7.635,148.590
C09807=1175.124,278.959,-68.356,-177.020,7.633,148.590
C09808=1175.127,278.711,-68.328,-177.022,7.630,148.590
C09809=1175.131,278.463,-68.298,-177.024,7.627,148.590
C09810=1175.137,278.214,-68.270,-177.027,7.624,148.590
C09811=1175.140,277.966,-68.241,-177.029,7.621,148.590
C09812=1175.144,277.717,-68.212,-177.032,7.618,148.590
C09813=1175.149,277.470,-68.183,-177.034,7.616,148.590
C09814=1175.154,277.221,-68.154,-177.037,7.613,148.590
C09815=1175.157,276.973,-68.126,-177.040,7.610,148.590
C09816=1175.162,276.725,-68.097,-177.043,7.607,148.590
C09817=1175.167,276.476,-68.068,-177.045,7.604,148.590
C09818=1175.170,276.228,-68.040,-177.047,7.602,148.591
C09819=1175.175,275.980,-68.011,-177.050,7.599,148.591
C09820=1175.179,275.731,-67.983,-177.053,7.596,148.591
C09821=1175.183,275.483,-67.954,-177.056,7.593,148.591
C09822=1175.188,275.235,-67.925,-177.058,7.590,148.591
C09823=1175.192,274.986,-67.897,-177.061,7.588,148.591
C09824=1175.196,274.738,-67.868,-177.063,7.585,148.591
C09825=1175.201,274.490,-67.839,-177.066,7.582,148.591
C09826=1175.205,274.241,-67.811,-177.069,7.579,148.591
C09827=1175.209,273.993,-67.782,-177.071,7.577,148.591
C09828=1175.214,273.745,-67.754,-177.074,7.574,148.591
C09829=1175.218,273.496,-67.725,-177.076,7.571,148.591
C09830=1175.222,273.248,-67.697,-177.079,7.568,148.591
C09831=1175.227,272.999,-67.669,-177.082,7.565,148.591
C09832=1175.231,272.751,-67.639,-177.084,7.563,148.591
C09833=1175.235,272.503,-67.611,-177.087,7.560,148.591
C09834=1175.240,272.254,-67.583,-177.090,7.557,148.591
C09835=1175.244,272.007,-67.555,-177.092,7.554,148.591
C09836=1175.249,271.758,-67.526,-177.094,7.552,148.591
C09837=1175.253,271.510,-67.498,-177.097,7.549,148.592
C09838=1175.257,271.261,-67.469,-177.100,7.546,148.592
C09839=1175.261,271.013,-67.441,-177.103,7.543,148.592
C09840=1175.266,270.765,-67.412,-177.105,7.541,148.592
C09841=1175.270,270.516,-67.384,-177.108,7.538,148.592
C09842=1175.275,270.268,-67.356,-177.110,7.535,148.592
C09843=1175.279,270.019,-67.328,-177.113,7.532,148.592
C09844=1175.283,269.772,-67.300,-177.115,7.530,148.592
C09845=1175.288,269.523,-67.271,-177.118,7.527,148.592
C09846=1175.292,269.275,-67.243,-177.121,7.524,148.592
C09847=1175.296,269.026,-67.215,-177.123,7.521,148.592
C09848=1175.301,268.778,-67.187,-177.126,7.518,148.592
C09849=1175.305,268.529,-67.158,-177.129,7.516,148.592
C09850=1175.310,268.281,-67.130,-177.132,7.513,148.592
C09851=1175.313,268.033,-67.102,-177.134,7.510,148.593
C09852=1175.318,267.784,-67.074,-177.137,7.508,148.593
C09853=1175.322,267.536,-67.046,-177.139,7.505,148.593
C09854=1175.327,267.288,-67.017,-177.142,7.502,148.593
C09855=1175.331,267.039,-66.989,-177.145,7.499,148.593
C09856=1175.336,266.791,-66.962,-177.147,7.497,148.593
C09857=1175.340,266.542,-66.933,-177.150,7.494,148.593
C09858=1175.345,266.294,-66.906,-177.152,7.491,148.593
C09859=1175.348,266.045,-66.878,-177.155,7.488,148.593
C09860=1175.353,265.797,-66.849,-177.157,7.486,148.593
C09861=1175.358,265.549,-66.821,-177.160,7.483,148.593
C09862=1175.362,265.300,-66.794,-177.163,7.480,148.593
C09863=1175.366,265.052,-66.766,-177.166,7.477,148.593
C09864=1175.371,264.803,-66.737,-177.168,7.475,148.594
C09865=1175.375,264.555,-66.710,-177.171,7.472,148.594
C09866=1175.379,264.308,-66.682,-177.174,7.469,148.594
C09867=1175.384,264.058,-66.654,-177.176,7.467,148.594
C09868=1175.388,263.810,-66.626,-177.179,7.464,148.594
C09869=1175.392,263.562,-66.598,-177.181,7.461,148.594
C09870=1175.397,263.313,-66.571,-177.184,7.458,148.594
C09871=1175.401,263.065,-66.543,-177.186,7.456,148.594
C09872=1175.406,262.816,-66.514,-177.189,7.453,148.594
C09873=1175.410,262.543,-66.484,-177.192,7.450,148.594
C09874=1175.416,262.270,-66.453,-177.195,7.447,148.594
C09875=1175.420,261.997,-66.423,-177.198,7.444,148.594
C09876=1175.425,261.725,-66.393,-177.200,7.441,148.594
C09877=1175.429,261.476,-66.364,-177.203,7.438,148.595
C09878=1175.434,261.227,-66.337,-177.206,7.435,148.595
C09879=1175.438,260.979,-66.309,-177.209,7.433,148.595
C09880=1175.442,260.730,-66.282,-177.211,7.430,148.595
C09881=1175.447,260.482,-66.254,-177.214,7.427,148.595
C09882=1175.451,260.233,-66.227,-177.216,7.425,148.595
C09883=1175.455,259.985,-66.199,-177.219,7.422,148.595
C09884=1175.460,259.737,-66.172,-177.222,7.419,148.595
C09885=1175.464,259.488,-66.143,-177.224,7.416,148.595
C09886=1175.469,259.239,-66.116,-177.227,7.415,148.596
C09887=1175.473,258.992,-66.088,-177.230,7.412,148.596
C09888=1175.478,258.743,-66.061,-177.233,7.409,148.596
C09889=1175.482,258.494,-66.033,-177.235,7.406,148.596
C09890=1175.486,258.246,-66.006,-177.237,7.403,148.596
C09891=1175.491,257.998,-65.978,-177.240,7.401,148.596
C09892=1175.495,257.749,-65.951,-177.243,7.399,148.596
C09893=1175.499,257.501,-65.923,-177.246,7.396,148.596
C09894=1175.504,257.253,-65.896,-177.248,7.393,148.596
C09895=1175.508,257.004,-65.869,-177.251,7.391,148.596
C09896=1175.512,256.755,-65.841,-177.253,7.388,148.596
C09897=1175.517,256.507,-65.814,-177.256,7.385,148.596
C09898=1175.522,256.258,-65.787,-177.259,7.383,148.597
C09899=1175.526,256.011,-65.759,-177.261,7.380,148.597
C09900=1175.530,255.761,-65.732,-177.264,7.377,148.597
C09901=1175.535,255.513,-65.704,-177.266,7.375,148.597
C09902=1175.539,255.265,-65.677,-177.269,7.372,148.597
C09903=1175.544,255.017,-65.650,-177.272,7.369,148.597
C09904=1175.548,254.767,-65.622,-177.274,7.367,148.597
C09905=1175.552,254.519,-65.595,-177.277,7.364,148.597
C09906=1175.557,254.271,-65.567,-177.280,7.361,148.598
C09907=1175.561,254.022,-65.540,-177.282,7.359,148.598
C09908=1175.566,253.774,-65.513,-177.285,7.356,148.598
C09909=1175.570,253.525,-65.486,-177.288,7.353,148.598
C09910=1175.574,253.277,-65.459,-177.290,7.351,148.598
C09911=1175.578,253.029,-65.432,-177.293,7.348,148.598
C09912=1175.583,252.780,-65.405,-177.296,7.345,148.598
C09913=1175.588,252.532,-65.377,-177.298,7.343,148.599
C09914=1175.592,252.283,-65.350,-177.301,7.340,148.599
C09915=1175.596,252.034,-65.323,-177.303,7.338,148.599
C09916=1175.601,251.786,-65.296,-177.306,7.335,148.599
C09917=1175.605,251.538,-65.269,-177.309,7.332,148.599
C09918=1175.609,251.289,-65.242,-177.311,7.331,148.599
C09919=1175.614,251.041,-65.215,-177.314,7.328,148.599
C09920=1175.619,250.792,-65.188,-177.317,7.325,148.599
C09921=1175.623,250.543,-65.160,-177.319,7.322,148.599
C09922=1175.627,250.295,-65.134,-177.322,7.320,148.600
C09923=1175.631,250.047,-65.107,-177.325,7.318,148.600
C09924=1175.636,249.798,-65.080,-177.327,7.315,148.600
C09925=1175.640,249.550,-65.052,-177.330,7.312,148.600
C09926=1175.645,249.301,-65.025,-177.333,7.310,148.600
C09927=1175.649,249.053,-64.999,-177.335,7.307,148.600
C09928=1175.654,248.804,-64.972,-177.338,7.304,148.600
C09929=1175.658,248.556,-64.945,-177.340,7.302,148.600
C09930=1175.662,248.307,-64.917,-177.344,7.299,148.601
C09931=1175.666,248.059,-64.891,-177.346,7.297,148.601
C09932=1175.671,247.810,-64.864,-177.348,7.294,148.601
C09933=1175.676,247.562,-64.837,-177.351,7.291,148.601
C09934=1175.680,247.313,-64.811,-177.354,7.289,148.601
C09935=1175.685,247.064,-64.784,-177.357,7.286,148.601
C09936=1175.689,246.816,-64.757,-177.359,7.284,148.601
C09937=1175.693,246.568,-64.730,-177.362,7.282,148.602
C09938=1175.698,246.319,-64.703,-177.365,7.279,148.602
C09939=1175.702,246.071,-64.676,-177.367,7.276,148.602
C09940=1175.707,245.822,-64.651,-177.370,7.274,148.602
C09941=1175.711,245.573,-64.624,-177.372,7.272,148.602
C09942=1175.716,245.325,-64.596,-177.375,7.269,148.602
C09943=1175.720,245.077,-64.570,-177.378,7.266,148.602
C09944=1175.725,244.828,-64.543,-177.380,7.264,148.603
C09945=1175.730,244.579,-64.517,-177.383,7.261,148.603
C09946=1175.733,244.331,-64.490,-177.385,7.259,148.603
C09947=1175.738,244.082,-64.463,-177.389,7.256,148.603
C09948=1175.742,243.834,-64.437,-177.391,7.253,148.603
C09949=1175.747,243.585,-64.410,-177.394,7.251,148.603
C09950=1175.751,243.337,-64.384,-177.397,7.248,148.604
C09951=1175.756,243.088,-64.357,-177.399,7.246,148.604
C09952=1175.761,242.839,-64.330,-177.402,7.243,148.604
C09953=1175.764,242.591,-64.304,-177.404,7.241,148.604
C09954=1175.769,242.343,-64.277,-177.407,7.239,148.604
C09955=1175.773,242.094,-64.251,-177.410,7.236,148.604
C09956=1175.778,241.845,-64.224,-177.412,7.234,148.604
C09957=1175.782,241.596,-64.198,-177.415,7.231,148.605
C09958=1175.787,241.348,-64.171,-177.417,7.229,148.605
C09959=1175.791,241.100,-64.145,-177.420,7.226,148.605
C09960=1175.796,240.851,-64.118,-177.423,7.224,148.605
C09961=1175.800,240.602,-64.092,-177.426,7.221,148.605
C09962=1175.805,240.353,-64.066,-177.428,7.219,148.605
C09963=1175.809,240.105,-64.039,-177.431,7.216,148.605
C09964=1175.813,239.856,-64.013,-177.434,7.213,148.606
C09965=1175.817,239.608,-63.986,-177.436,7.211,148.606
C09966=1175.822,239.360,-63.961,-177.439,7.208,148.606
C09967=1175.827,239.111,-63.934,-177.441,7.206,148.606
C09968=1175.831,238.862,-63.908,-177.444,7.204,148.606
C09969=1175.836,238.614,-63.881,-177.447,7.202,148.606
C09970=1175.840,238.365,-63.855,-177.449,7.199,148.607
C09971=1175.844,238.117,-63.829,-177.452,7.197,148.607
C09972=1175.849,237.868,-63.802,-177.455,7.194,148.607
C09973=1175.853,237.619,-63.777,-177.457,7.192,148.607
C09974=1175.858,237.371,-63.750,-177.460,7.189,148.607
C09975=1175.863,237.122,-63.724,-177.462,7.187,148.607
C09976=1175.867,236.874,-63.698,-177.466,7.184,148.608
C09977=1175.872,236.602,-63.669,-177.468,7.181,148.608
C09978=1175.876,236.331,-63.640,-177.472,7.179,148.608
C09979=1175.881,236.059,-63.612,-177.474,7.176,148.608
C09980=1175.886,235.787,-63.583,-177.477,7.174,148.608
C09981=1175.890,235.538,-63.557,-177.480,7.171,148.609
C09982=1175.895,235.290,-63.532,-177.482,7.169,148.609
C09983=1175.900,235.041,-63.506,-177.485,7.166,148.609
C09984=1175.904,234.793,-63.479,-177.487,7.164,148.609
C09985=1175.908,234.544,-63.453,-177.491,7.161,148.609
C09986=1175.913,234.295,-63.428,-177.493,7.158,148.609
C09987=1175.918,234.047,-63.402,-177.496,7.157,148.610
C09988=1175.922,233.799,-63.375,-177.499,7.154,148.610
C09989=1175.926,233.550,-63.349,-177.501,7.152,148.610
C09990=1175.930,233.301,-63.324,-177.504,7.149,148.610
C09991=1175.935,233.052,-63.297,-177.506,7.147,148.610
C09992=1175.940,232.804,-63.272,-177.510,7.144,148.611
C09993=1175.944,232.556,-63.245,-177.512,7.142,148.611
C09994=1175.948,232.307,-63.220,-177.515,7.139,148.611
C09995=1175.953,232.058,-63.194,-177.517,7.137,148.611
C09996=1175.958,231.810,-63.168,-177.520,7.135,148.611
//INST
///DATE 2021/06/15 17:25
///ATTR SC,RW,RJ
////FRAME ROBOT
///GROUP1 RB1
NOP
MOVL C00000 V=800.0 PL=0
MOVL C00001 V=800.0 PL=0
MOVL C00002 V=800.0 PL=0
MOVL C00003 V=800.0 PL=0
MOVL C00004 V=800.0 PL=0
MOVL C00005 V=800.0 PL=0
MOVL C00006 V=800.0 PL=0
MOVL C00007 V=800.0 PL=0
MOVL C00008 V=800.0 PL=0
MOVL C00009 V=800.0 PL=0
MOVL C00010 V=800.0 PL=0
MOVL C00011 V=800.0 PL=0
MOVL C00012 V=800.0 PL=0
MOVL C00013 V=800.0 PL=0
MOVL C00014 V=800.0 PL=0
MOVL C00015 V=800.0 PL=0
MOVL C00016 V=800.0 PL=0
MOVL C00017 V=800.0 PL=0
MOVL C00018 V=800.0 PL=0
MOVL C00019 V=800.0 PL=0
MOVL C00020 V=800.0 PL=0
MOVL C00021 V=800.0 PL=0
MOVL C00022 V=800.0 PL=0
MOVL C00023 V=800.0 PL=0
MOVL C00024 V=800.0 PL=0
MOVL C00025 V=800.0 PL=0
MOVL C00026 V=800.0 PL=0
MOVL C00027 V=800.0 PL=0
MOVL C00028 V=800.0 PL=0
MOVL C00029 V=800.0 PL=0
MOVL C00030 V=800.0 PL=0
MOVL C00031 V=800.0 PL=0
MOVL C00032 V=800.0 PL=0
MOVL C00033 V=800.0 PL=0
MOVL C00034 V=800.0 PL=0
MOVL C00035 V=800.0 PL=0
MOVL C00036 V=800.0 PL=0
MOVL C00037 V=800.0 PL=0
MOVL C00038 V=800.0 PL=0
MOVL C00039 V=800.0 PL=0
MOVL C00040 V=800.0 PL=0
MOVL C00041 V=800.0 PL=0
MOVL C00042 V=800.0 PL=0
MOVL C00043 V=800.0 PL=0
MOVL C00044 V=800.0 PL=0
MOVL C00045 V=800.0 PL=0
MOVL C00046 V=800.0 PL=0
MOVL C00047 V=800.0 PL=0
MOVL C00048 V=800.0 PL=0
MOVL C00049 V=800.0 PL=0
MOVL C00050 V=800.0 PL=0
MOVL C00051 V=800.0 PL=0
MOVL C00052 V=800.0 PL=0
MOVL C00053 V=800.0 PL=0
MOVL C00054 V=800.0 PL=0
MOVL C00055 V=800.0 PL=0
MOVL C00056 V=800.0 PL=0
MOVL C00057 V=800.0 PL=0
MOVL C00058 V=800.0 PL=0
MOVL C00059 V=800.0 PL=0
MOVL C00060 V=800.0 PL=0
MOVL C00061 V=800.0 PL=0
MOVL C00062 V=800.0 PL=0
MOVL C00063 V=800.0 PL=0
MOVL C00064 V=800.0 PL=0
MOVL C00065 V=800.0 PL=0
MOVL C00066 V=800.0 PL=0
MOVL C00067 V=800.0 PL=0
MOVL C00068 V=800.0 PL=0
MOVL C00069 V=800.0 PL=0
MOVL C00070 V=800.0 PL=0
MOVL C00071 V=800.0 PL=0
MOVL C00072 V=800.0 PL=0
MOVL C00073 V=800.0 PL=0
MOVL C00074 V=800.0 PL=0
MOVL C00075 V=800.0 PL=0
MOVL C00076 V=800.0 PL=0
MOVL C00077 V=800.0 PL=0
MOVL C00078 V=800.0 PL=0
MOVL C00079 V=800.0 PL=0
MOVL C00080 V=800.0 PL=0
MOVL C00081 V=800.0 PL=0
MOVL C00082 V=800.0 PL=0
MOVL C00083 V=800.0 PL=0
MOVL C00084 V=800.0 PL=0
MOVL C00085 V=800.0 PL=0
MOVL C00086 V=800.0 PL=0
MOVL C00087 V=800.0 PL=0
MOVL C00088 V=800.0 PL=0
MOVL C00089 V=800.0 PL=0
MOVL C00090 V=800.0 PL=0
MOVL C00091 V=800.0 PL=0
MOVL C00092 V=800.0 PL=0
MOVL C00093 V=800.0 PL=0
MOVL C00094 V=800.0 PL=0
MOVL C00095 V=800.0 PL=0
MOVL C00096 V=800.0 PL=0
MOVL C00097 V=800.0 PL=0
MOVL C00098 V=800.0 PL=0
MOVL C00099 V=800.0 PL=0
MOVL C00100 V=800.0 PL=0
MOVL C00101 V=800.0 PL=0
MOVL C00102 V=800.0 PL=0
MOVL C00103 V=800.0 PL=0
MOVL C00104 V=800.0 PL=0
MOVL C00105 V=800.0 PL=0
MOVL C00106 V=800.0 PL=0
MOVL C00107 V=800.0 PL=0
MOVL C00108 V=800.0 PL=0
MOVL C00109 V=800.0 PL=0
MOVL C00110 V=800.0 PL=0
MOVL C00111 V=800.0 PL=0
MOVL C00112 V=800.0 PL=0
MOVL C00113 V=800.0 PL=0
MOVL C00114 V=800.0 PL=0
MOVL C00115 V=800.0 PL=0
MOVL C00116 V=800.0 PL=0
MOVL C00117 V=800.0 PL=0
MOVL C00118 V=800.0 PL=0
MOVL C00119 V=800.0 PL=0
MOVL C00120 V=800.0 PL=0
MOVL C00121 V=800.0 PL=0
MOVL C00122 V=800.0 PL=0
MOVL C00123 V=800.0 PL=0
MOVL C00124 V=800.0 PL=0
MOVL C00125 V=800.0 PL=0
MOVL C00126 V=800.0 PL=0
MOVL C00127 V=800.0 PL=0
MOVL C00128 V=800.0 PL=0
MOVL C00129 V=800.0 PL=0
MOVL C00130 V=800.0 PL=0
MOVL C00131 V=800.0 PL=0
MOVL C00132 V=800.0 PL=0
MOVL C00133 V=800.0 PL=0
MOVL C00134 V=800.0 PL=0
MOVL C00135 V=800.0 PL=0
MOVL C00136 V=800.0 PL=0
MOVL C00137 V=800.0 PL=0
MOVL C00138 V=800.0 PL=0
MOVL C00139 V=800.0 PL=0
MOVL C00140 V=800.0 PL=0
MOVL C00141 V=800.0 PL=0
MOVL C00142 V=800.0 PL=0
MOVL C00143 V=800.0 PL=0
MOVL C00144 V=800.0 PL=0
MOVL C00145 V=800.0 PL=0
MOVL C00146 V=800.0 PL=0
MOVL C00147 V=800.0 PL=0
MOVL C00148 V=800.0 PL=0
MOVL C00149 V=800.0 PL=0
MOVL C00150 V=800.0 PL=0
MOVL C00151 V=800.0 PL=0
MOVL C00152 V=800.0 PL=0
MOVL C00153 V=800.0 PL=0
MOVL C00154 V=800.0 PL=0
MOVL C00155 V=800.0 PL=0
MOVL C00156 V=800.0 PL=0
MOVL C00157 V=800.0 PL=0
MOVL C00158 V=800.0 PL=0
MOVL C00159 V=800.0 PL=0
MOVL C00160 V=800.0 PL=0
MOVL C00161 V=800.0 PL=0
MOVL C00162 V=800.0 PL=0
MOVL C00163 V=800.0 PL=0
MOVL C00164 V=800.0 PL=0
MOVL C00165 V=800.0 PL=0
MOVL C00166 V=800.0 PL=0
MOVL C00167 V=800.0 PL=0
MOVL C00168 V=800.0 PL=0
MOVL C00169 V=800.0 PL=0
MOVL C00170 V=800.0 PL=0
MOVL C00171 V=800.0 PL=0
MOVL C00172 V=800.0 PL=0
MOVL C00173 V=800.0 PL=0
MOVL C00174 V=800.0 PL=0
MOVL C00175 V=800.0 PL=0
MOVL C00176 V=800.0 PL=0
MOVL C00177 V=800.0 PL=0
MOVL C00178 V=800.0 PL=0
MOVL C00179 V=800.0 PL=0
MOVL C00180 V=800.0 PL=0
MOVL C00181 V=800.0 PL=0
MOVL C00182 V=800.0 PL=0
MOVL C00183 V=800.0 PL=0
MOVL C00184 V=800.0 PL=0
MOVL C00185 V=800.0 PL=0
MOVL C00186 V=800.0 PL=0
MOVL C00187 V=800.0 PL=0
MOVL C00188 V=800.0 PL=0
MOVL C00189 V=800.0 PL=0
MOVL C00190 V=800.0 PL=0
MOVL C00191 V=800.0 PL=0
MOVL C00192 V=800.0 PL=0
MOVL C00193 V=800.0 PL=0
MOVL C00194 V=800.0 PL=0
MOVL C00195 V=800.0 PL=0
MOVL C00196 V=800.0 PL=0
MOVL C00197 V=800.0 PL=0
MOVL C00198 V=800.0 PL=0
MOVL C00199 V=800.0 PL=0
MOVL C00200 V=800.0 PL=0
MOVL C00201 V=800.0 PL=0
MOVL C00202 V=800.0 PL=0
MOVL C00203 V=800.0 PL=0
MOVL C00204 V=800.0 PL=0
MOVL C00205 V=800.0 PL=0
MOVL C00206 V=800.0 PL=0
MOVL C00207 V=800.0 PL=0
MOVL C00208 V=800.0 PL=0
MOVL C00209 V=800.0 PL=0
MOVL C00210 V=800.0 PL=0
MOVL C00211 V=800.0 PL=0
MOVL C00212 V=800.0 PL=0
MOVL C00213 V=800.0 PL=0
MOVL C00214 V=800.0 PL=0
MOVL C00215 V=800.0 PL=0
MOVL C00216 V=800.0 PL=0
MOVL C00217 V=800.0 PL=0
MOVL C00218 V=800.0 PL=0
MOVL C00219 V=800.0 PL=0
MOVL C00220 V=800.0 PL=0
MOVL C00221 V=800.0 PL=0
MOVL C00222 V=800.0 PL=0
MOVL C00223 V=800.0 PL=0
MOVL C00224 V=800.0 PL=0
MOVL C00225 V=800.0 PL=0
MOVL C00226 V=800.0 PL=0
MOVL C00227 V=800.0 PL=0
MOVL C00228 V=800.0 PL=0
MOVL C00229 V=800.0 PL=0
MOVL C00230 V=800.0 PL=0
MOVL C00231 V=800.0 PL=0
MOVL C00232 V=800.0 PL=0
MOVL C00233 V=800.0 PL=0
MOVL C00234 V=800.0 PL=0
MOVL C00235 V=800.0 PL=0
MOVL C00236 V=800.0 PL=0
MOVL C00237 V=800.0 PL=0
MOVL C00238 V=800.0 PL=0
MOVL C00239 V=800.0 PL=0
MOVL C00240 V=800.0 PL=0
MOVL C00241 V=800.0 PL=0
MOVL C00242 V=800.0 PL=0
MOVL C00243 V=800.0 PL=0
MOVL C00244 V=800.0 PL=0
MOVL C00245 V=800.0 PL=0
MOVL C00246 V=800.0 PL=0
MOVL C00247 V=800.0 PL=0
MOVL C00248 V=800.0 PL=0
MOVL C00249 V=800.0 PL=0
MOVL C00250 V=800.0 PL=0
MOVL C00251 V=800.0 PL=0
MOVL C00252 V=800.0 PL=0
MOVL C00253 V=800.0 PL=0
MOVL C00254 V=800.0 PL=0
MOVL C00255 V=800.0 PL=0
MOVL C00256 V=800.0 PL=0
MOVL C00257 V=800.0 PL=0
MOVL C00258 V=800.0 PL=0
MOVL C00259 V=800.0 PL=0
MOVL C00260 V=800.0 PL=0
MOVL C00261 V=800.0 PL=0
MOVL C00262 V=800.0 PL=0
MOVL C00263 V=800.0 PL=0
MOVL C00264 V=800.0 PL=0
MOVL C00265 V=800.0 PL=0
MOVL C00266 V=800.0 PL=0
MOVL C00267 V=800.0 PL=0
MOVL C00268 V=800.0 PL=0
MOVL C00269 V=800.0 PL=0
MOVL C00270 V=800.0 PL=0
MOVL C00271 V=800.0 PL=0
MOVL C00272 V=800.0 PL=0
MOVL C00273 V=800.0 PL=0
MOVL C00274 V=800.0 PL=0
MOVL C00275 V=800.0 PL=0
MOVL C00276 V=800.0 PL=0
MOVL C00277 V=800.0 PL=0
MOVL C00278 V=800.0 PL=0
MOVL C00279 V=800.0 PL=0
MOVL C00280 V=800.0 PL=0
MOVL C00281 V=800.0 PL=0
MOVL C00282 V=800.0 PL=0
MOVL C00283 V=800.0 PL=0
MOVL C00284 V=800.0 PL=0
MOVL C00285 V=800.0 PL=0
MOVL C00286 V=800.0 PL=0
MOVL C00287 V=800.0 PL=0
MOVL C00288 V=800.0 PL=0
MOVL C00289 V=800.0 PL=0
MOVL C00290 V=800.0 PL=0
MOVL C00291 V=800.0 PL=0
MOVL C00292 V=800.0 PL=0
MOVL C00293 V=800.0 PL=0
MOVL C00294 V=800.0 PL=0
MOVL C00295 V=800.0 PL=0
MOVL C00296 V=800.0 PL=0
MOVL C00297 V=800.0 PL=0
MOVL C00298 V=800.0 PL=0
MOVL C00299 V=800.0 PL=0
MOVL C00300 V=800.0 PL=0
MOVL C00301 V=800.0 PL=0
MOVL C00302 V=800.0 PL=0
MOVL C00303 V=800.0 PL=0
MOVL C00304 V=800.0 PL=0
MOVL C00305 V=800.0 PL=0
MOVL C00306 V=800.0 PL=0
MOVL C00307 V=800.0 PL=0
MOVL C00308 V=800.0 PL=0
MOVL C00309 V=800.0 PL=0
MOVL C00310 V=800.0 PL=0
MOVL C00311 V=800.0 PL=0
MOVL C00312 V=800.0 PL=0
MOVL C00313 V=800.0 PL=0
MOVL C00314 V=800.0 PL=0
MOVL C00315 V=800.0 PL=0
MOVL C00316 V=800.0 PL=0
MOVL C00317 V=800.0 PL=0
MOVL C00318 V=800.0 PL=0
MOVL C00319 V=800.0 PL=0
MOVL C00320 V=800.0 PL=0
MOVL C00321 V=800.0 PL=0
MOVL C00322 V=800.0 PL=0
MOVL C00323 V=800.0 PL=0
MOVL C00324 V=800.0 PL=0
MOVL C00325 V=800.0 PL=0
MOVL C00326 V=800.0 PL=0
MOVL C00327 V=800.0 PL=0
MOVL C00328 V=800.0 PL=0
MOVL C00329 V=800.0 PL=0
MOVL C00330 V=800.0 PL=0
MOVL C00331 V=800.0 PL=0
MOVL C00332 V=800.0 PL=0
MOVL C00333 V=800.0 PL=0
MOVL C00334 V=800.0 PL=0
MOVL C00335 V=800.0 PL=0
MOVL C00336 V=800.0 PL=0
MOVL C00337 V=800.0 PL=0
MOVL C00338 V=800.0 PL=0
MOVL C00339 V=800.0 PL=0
MOVL C00340 V=800.0 PL=0
MOVL C00341 V=800.0 PL=0
MOVL C00342 V=800.0 PL=0
MOVL C00343 V=800.0 PL=0
MOVL C00344 V=800.0 PL=0
MOVL C00345 V=800.0 PL=0
MOVL C00346 V=800.0 PL=0
MOVL C00347 V=800.0 PL=0
MOVL C00348 V=800.0 PL=0
MOVL C00349 V=800.0 PL=0
MOVL C00350 V=800.0 PL=0
MOVL C00351 V=800.0 PL=0
MOVL C00352 V=800.0 PL=0
MOVL C00353 V=800.0 PL=0
MOVL C00354 V=800.0 PL=0
MOVL C00355 V=800.0 PL=0
MOVL C00356 V=800.0 PL=0
MOVL C00357 V=800.0 PL=0
MOVL C00358 V=800.0 PL=0
MOVL C00359 V=800.0 PL=0
MOVL C00360 V=800.0 PL=0
MOVL C00361 V=800.0 PL=0
MOVL C00362 V=800.0 PL=0
MOVL C00363 V=800.0 PL=0
MOVL C00364 V=800.0 PL=0
MOVL C00365 V=800.0 PL=0
MOVL C00366 V=800.0 PL=0
MOVL C00367 V=800.0 PL=0
MOVL C00368 V=800.0 PL=0
MOVL C00369 V=800.0 PL=0
MOVL C00370 V=800.0 PL=0
MOVL C00371 V=800.0 PL=0
MOVL C00372 V=800.0 PL=0
MOVL C00373 V=800.0 PL=0
MOVL C00374 V=800.0 PL=0
MOVL C00375 V=800.0 PL=0
MOVL C00376 V=800.0 PL=0
MOVL C00377 V=800.0 PL=0
MOVL C00378 V=800.0 PL=0
MOVL C00379 V=800.0 PL=0
MOVL C00380 V=800.0 PL=0
MOVL C00381 V=800.0 PL=0
MOVL C00382 V=800.0 PL=0
MOVL C00383 V=800.0 PL=0
MOVL C00384 V=800.0 PL=0
MOVL C00385 V=800.0 PL=0
MOVL C00386 V=800.0 PL=0
MOVL C00387 V=800.0 PL=0
MOVL C00388 V=800.0 PL=0
MOVL C00389 V=800.0 PL=0
MOVL C00390 V=800.0 PL=0
MOVL C00391 V=800.0 PL=0
MOVL C00392 V=800.0 PL=0
MOVL C00393 V=800.0 PL=0
MOVL C00394 V=800.0 PL=0
MOVL C00395 V=800.0 PL=0
MOVL C00396 V=800.0 PL=0
MOVL C00397 V=800.0 PL=0
MOVL C00398 V=800.0 PL=0
MOVL C00399 V=800.0 PL=0
MOVL C00400 V=800.0 PL=0
MOVL C00401 V=800.0 PL=0
MOVL C00402 V=800.0 PL=0
MOVL C00403 V=800.0 PL=0
MOVL C00404 V=800.0 PL=0
MOVL C00405 V=800.0 PL=0
MOVL C00406 V=800.0 PL=0
MOVL C00407 V=800.0 PL=0
MOVL C00408 V=800.0 PL=0
MOVL C00409 V=800.0 PL=0
MOVL C00410 V=800.0 PL=0
MOVL C00411 V=800.0 PL=0
MOVL C00412 V=800.0 PL=0
MOVL C00413 V=800.0 PL=0
MOVL C00414 V=800.0 PL=0
MOVL C00415 V=800.0 PL=0
MOVL C00416 V=800.0 PL=0
MOVL C00417 V=800.0 PL=0
MOVL C00418 V=800.0 PL=0
MOVL C00419 V=800.0 PL=0
MOVL C00420 V=800.0 PL=0
MOVL C00421 V=800.0 PL=0
MOVL C00422 V=800.0 PL=0
MOVL C00423 V=800.0 PL=0
MOVL C00424 V=800.0 PL=0
MOVL C00425 V=800.0 PL=0
MOVL C00426 V=800.0 PL=0
MOVL C00427 V=800.0 PL=0
MOVL C00428 V=800.0 PL=0
MOVL C00429 V=800.0 PL=0
MOVL C00430 V=800.0 PL=0
MOVL C00431 V=800.0 PL=0
MOVL C00432 V=800.0 PL=0
MOVL C00433 V=800.0 PL=0
MOVL C00434 V=800.0 PL=0
MOVL C00435 V=800.0 PL=0
MOVL C00436 V=800.0 PL=0
MOVL C00437 V=800.0 PL=0
MOVL C00438 V=800.0 PL=0
MOVL C00439 V=800.0 PL=0
MOVL C00440 V=800.0 PL=0
MOVL C00441 V=800.0 PL=0
MOVL C00442 V=800.0 PL=0
MOVL C00443 V=800.0 PL=0
MOVL C00444 V=800.0 PL=0
MOVL C00445 V=800.0 PL=0
MOVL C00446 V=800.0 PL=0
MOVL C00447 V=800.0 PL=0
MOVL C00448 V=800.0 PL=0
MOVL C00449 V=800.0 PL=0
MOVL C00450 V=800.0 PL=0
MOVL C00451 V=800.0 PL=0
MOVL C00452 V=800.0 PL=0
MOVL C00453 V=800.0 PL=0
MOVL C00454 V=800.0 PL=0
MOVL C00455 V=800.0 PL=0
MOVL C00456 V=800.0 PL=0
MOVL C00457 V=800.0 PL=0
MOVL C00458 V=800.0 PL=0
MOVL C00459 V=800.0 PL=0
MOVL C00460 V=800.0 PL=0
MOVL C00461 V=800.0 PL=0
MOVL C00462 V=800.0 PL=0
MOVL C00463 V=800.0 PL=0
MOVL C00464 V=800.0 PL=0
MOVL C00465 V=800.0 PL=0
MOVL C00466 V=800.0 PL=0
MOVL C00467 V=800.0 PL=0
MOVL C00468 V=800.0 PL=0
MOVL C00469 V=800.0 PL=0
MOVL C00470 V=800.0 PL=0
MOVL C00471 V=800.0 PL=0
MOVL C00472 V=800.0 PL=0
MOVL C00473 V=800.0 PL=0
MOVL C00474 V=800.0 PL=0
MOVL C00475 V=800.0 PL=0
MOVL C00476 V=800.0 PL=0
MOVL C00477 V=800.0 PL=0
MOVL C00478 V=800.0 PL=0
MOVL C00479 V=800.0 PL=0
MOVL C00480 V=800.0 PL=0
MOVL C00481 V=800.0 PL=0
MOVL C00482 V=800.0 PL=0
MOVL C00483 V=800.0 PL=0
MOVL C00484 V=800.0 PL=0
MOVL C00485 V=800.0 PL=0
MOVL C00486 V=800.0 PL=0
MOVL C00487 V=800.0 PL=0
MOVL C00488 V=800.0 PL=0
MOVL C00489 V=800.0 PL=0
MOVL C00490 V=800.0 PL=0
MOVL C00491 V=800.0 PL=0
MOVL C00492 V=800.0 PL=0
MOVL C00493 V=800.0 PL=0
MOVL C00494 V=800.0 PL=0
MOVL C00495 V=800.0 PL=0
MOVL C00496 V=800.0 PL=0
MOVL C00497 V=800.0 PL=0
MOVL C00498 V=800.0 PL=0
MOVL C00499 V=800.0 PL=0
MOVL C00500 V=800.0 PL=0
MOVL C00501 V=800.0 PL=0
MOVL C00502 V=800.0 PL=0
MOVL C00503 V=800.0 PL=0
MOVL C00504 V=800.0 PL=0
MOVL C00505 V=800.0 PL=0
MOVL C00506 V=800.0 PL=0
MOVL C00507 V=800.0 PL=0
MOVL C00508 V=800.0 PL=0
MOVL C00509 V=800.0 PL=0
MOVL C00510 V=800.0 PL=0
MOVL C00511 V=800.0 PL=0
MOVL C00512 V=800.0 PL=0
MOVL C00513 V=800.0 PL=0
MOVL C00514 V=800.0 PL=0
MOVL C00515 V=800.0 PL=0
MOVL C00516 V=800.0 PL=0
MOVL C00517 V=800.0 PL=0
MOVL C00518 V=800.0 PL=0
MOVL C00519 V=800.0 PL=0
MOVL C00520 V=800.0 PL=0
MOVL C00521 V=800.0 PL=0
MOVL C00522 V=800.0 PL=0
MOVL C00523 V=800.0 PL=0
MOVL C00524 V=800.0 PL=0
MOVL C00525 V=800.0 PL=0
MOVL C00526 V=800.0 PL=0
MOVL C00527 V=800.0 PL=0
MOVL C00528 V=800.0 PL=0
MOVL C00529 V=800.0 PL=0
MOVL C00530 V=800.0 PL=0
MOVL C00531 V=800.0 PL=0
MOVL C00532 V=800.0 PL=0
MOVL C00533 V=800.0 PL=0
MOVL C00534 V=800.0 PL=0
MOVL C00535 V=800.0 PL=0
MOVL C00536 V=800.0 PL=0
MOVL C00537 V=800.0 PL=0
MOVL C00538 V=800.0 PL=0
MOVL C00539 V=800.0 PL=0
MOVL C00540 V=800.0 PL=0
MOVL C00541 V=800.0 PL=0
MOVL C00542 V=800.0 PL=0
MOVL C00543 V=800.0 PL=0
MOVL C00544 V=800.0 PL=0
MOVL C00545 V=800.0 PL=0
MOVL C00546 V=800.0 PL=0
MOVL C00547 V=800.0 PL=0
MOVL C00548 V=800.0 PL=0
MOVL C00549 V=800.0 PL=0
MOVL C00550 V=800.0 PL=0
MOVL C00551 V=800.0 PL=0
MOVL C00552 V=800.0 PL=0
MOVL C00553 V=800.0 PL=0
MOVL C00554 V=800.0 PL=0
MOVL C00555 V=800.0 PL=0
MOVL C00556 V=800.0 PL=0
MOVL C00557 V=800.0 PL=0
MOVL C00558 V=800.0 PL=0
MOVL C00559 V=800.0 PL=0
MOVL C00560 V=800.0 PL=0
MOVL C00561 V=800.0 PL=0
MOVL C00562 V=800.0 PL=0
MOVL C00563 V=800.0 PL=0
MOVL C00564 V=800.0 PL=0
MOVL C00565 V=800.0 PL=0
MOVL C00566 V=800.0 PL=0
MOVL C00567 V=800.0 PL=0
MOVL C00568 V=800.0 PL=0
MOVL C00569 V=800.0 PL=0
MOVL C00570 V=800.0 PL=0
MOVL C00571 V=800.0 PL=0
MOVL C00572 V=800.0 PL=0
MOVL C00573 V=800.0 PL=0
MOVL C00574 V=800.0 PL=0
MOVL C00575 V=800.0 PL=0
MOVL C00576 V=800.0 PL=0
MOVL C00577 V=800.0 PL=0
MOVL C00578 V=800.0 PL=0
MOVL C00579 V=800.0 PL=0
MOVL C00580 V=800.0 PL=0
MOVL C00581 V=800.0 PL=0
MOVL C00582 V=800.0 PL=0
MOVL C00583 V=800.0 PL=0
MOVL C00584 V=800.0 PL=0
MOVL C00585 V=800.0 PL=0
MOVL C00586 V=800.0 PL=0
MOVL C00587 V=800.0 PL=0
MOVL C00588 V=800.0 PL=0
MOVL C00589 V=800.0 PL=0
MOVL C00590 V=800.0 PL=0
MOVL C00591 V=800.0 PL=0
MOVL C00592 V=800.0 PL=0
MOVL C00593 V=800.0 PL=0
MOVL C00594 V=800.0 PL=0
MOVL C00595 V=800.0 PL=0
MOVL C00596 V=800.0 PL=0
MOVL C00597 V=800.0 PL=0
MOVL C00598 V=800.0 PL=0
MOVL C00599 V=800.0 PL=0
MOVL C00600 V=800.0 PL=0
MOVL C00601 V=800.0 PL=0
MOVL C00602 V=800.0 PL=0
MOVL C00603 V=800.0 PL=0
MOVL C00604 V=800.0 PL=0
MOVL C00605 V=800.0 PL=0
MOVL C00606 V=800.0 PL=0
MOVL C00607 V=800.0 PL=0
MOVL C00608 V=800.0 PL=0
MOVL C00609 V=800.0 PL=0
MOVL C00610 V=800.0 PL=0
MOVL C00611 V=800.0 PL=0
MOVL C00612 V=800.0 PL=0
MOVL C00613 V=800.0 PL=0
MOVL C00614 V=800.0 PL=0
MOVL C00615 V=800.0 PL=0
MOVL C00616 V=800.0 PL=0
MOVL C00617 V=800.0 PL=0
MOVL C00618 V=800.0 PL=0
MOVL C00619 V=800.0 PL=0
MOVL C00620 V=800.0 PL=0
MOVL C00621 V=800.0 PL=0
MOVL C00622 V=800.0 PL=0
MOVL C00623 V=800.0 PL=0
MOVL C00624 V=800.0 PL=0
MOVL C00625 V=800.0 PL=0
MOVL C00626 V=800.0 PL=0
MOVL C00627 V=800.0 PL=0
MOVL C00628 V=800.0 PL=0
MOVL C00629 V=800.0 PL=0
MOVL C00630 V=800.0 PL=0
MOVL C00631 V=800.0 PL=0
MOVL C00632 V=800.0 PL=0
MOVL C00633 V=800.0 PL=0
MOVL C00634 V=800.0 PL=0
MOVL C00635 V=800.0 PL=0
MOVL C00636 V=800.0 PL=0
MOVL C00637 V=800.0 PL=0
MOVL C00638 V=800.0 PL=0
MOVL C00639 V=800.0 PL=0
MOVL C00640 V=800.0 PL=0
MOVL C00641 V=800.0 PL=0
MOVL C00642 V=800.0 PL=0
MOVL C00643 V=800.0 PL=0
MOVL C00644 V=800.0 PL=0
MOVL C00645 V=800.0 PL=0
MOVL C00646 V=800.0 PL=0
MOVL C00647 V=800.0 PL=0
MOVL C00648 V=800.0 PL=0
MOVL C00649 V=800.0 PL=0
MOVL C00650 V=800.0 PL=0
MOVL C00651 V=800.0 PL=0
MOVL C00652 V=800.0 PL=0
MOVL C00653 V=800.0 PL=0
MOVL C00654 V=800.0 PL=0
MOVL C00655 V=800.0 PL=0
MOVL C00656 V=800.0 PL=0
MOVL C00657 V=800.0 PL=0
MOVL C00658 V=800.0 PL=0
MOVL C00659 V=800.0 PL=0
MOVL C00660 V=800.0 PL=0
MOVL C00661 V=800.0 PL=0
MOVL C00662 V=800.0 PL=0
MOVL C00663 V=800.0 PL=0
MOVL C00664 V=800.0 PL=0
MOVL C00665 V=800.0 PL=0
MOVL C00666 V=800.0 PL=0
MOVL C00667 V=800.0 PL=0
MOVL C00668 V=800.0 PL=0
MOVL C00669 V=800.0 PL=0
MOVL C00670 V=800.0 PL=0
MOVL C00671 V=800.0 PL=0
MOVL C00672 V=800.0 PL=0
MOVL C00673 V=800.0 PL=0
MOVL C00674 V=800.0 PL=0
MOVL C00675 V=800.0 PL=0
MOVL C00676 V=800.0 PL=0
MOVL C00677 V=800.0 PL=0
MOVL C00678 V=800.0 PL=0
MOVL C00679 V=800.0 PL=0
MOVL C00680 V=800.0 PL=0
MOVL C00681 V=800.0 PL=0
MOVL C00682 V=800.0 PL=0
MOVL C00683 V=800.0 PL=0
MOVL C00684 V=800.0 PL=0
MOVL C00685 V=800.0 PL=0
MOVL C00686 V=800.0 PL=0
MOVL C00687 V=800.0 PL=0
MOVL C00688 V=800.0 PL=0
MOVL C00689 V=800.0 PL=0
MOVL C00690 V=800.0 PL=0
MOVL C00691 V=800.0 PL=0
MOVL C00692 V=800.0 PL=0
MOVL C00693 V=800.0 PL=0
MOVL C00694 V=800.0 PL=0
MOVL C00695 V=800.0 PL=0
MOVL C00696 V=800.0 PL=0
MOVL C00697 V=800.0 PL=0
MOVL C00698 V=800.0 PL=0
MOVL C00699 V=800.0 PL=0
MOVL C00700 V=800.0 PL=0
MOVL C00701 V=800.0 PL=0
MOVL C00702 V=800.0 PL=0
MOVL C00703 V=800.0 PL=0
MOVL C00704 V=800.0 PL=0
MOVL C00705 V=800.0 PL=0
MOVL C00706 V=800.0 PL=0
MOVL C00707 V=800.0 PL=0
MOVL C00708 V=800.0 PL=0
MOVL C00709 V=800.0 PL=0
MOVL C00710 V=800.0 PL=0
MOVL C00711 V=800.0 PL=0
MOVL C00712 V=800.0 PL=0
MOVL C00713 V=800.0 PL=0
MOVL C00714 V=800.0 PL=0
MOVL C00715 V=800.0 PL=0
MOVL C00716 V=800.0 PL=0
MOVL C00717 V=800.0 PL=0
MOVL C00718 V=800.0 PL=0
MOVL C00719 V=800.0 PL=0
MOVL C00720 V=800.0 PL=0
MOVL C00721 V=800.0 PL=0
MOVL C00722 V=800.0 PL=0
MOVL C00723 V=800.0 PL=0
MOVL C00724 V=800.0 PL=0
MOVL C00725 V=800.0 PL=0
MOVL C00726 V=800.0 PL=0
MOVL C00727 V=800.0 PL=0
MOVL C00728 V=800.0 PL=0
MOVL C00729 V=800.0 PL=0
MOVL C00730 V=800.0 PL=0
MOVL C00731 V=800.0 PL=0
MOVL C00732 V=800.0 PL=0
MOVL C00733 V=800.0 PL=0
MOVL C00734 V=800.0 PL=0
MOVL C00735 V=800.0 PL=0
MOVL C00736 V=800.0 PL=0
MOVL C00737 V=800.0 PL=0
MOVL C00738 V=800.0 PL=0
MOVL C00739 V=800.0 PL=0
MOVL C00740 V=800.0 PL=0
MOVL C00741 V=800.0 PL=0
MOVL C00742 V=800.0 PL=0
MOVL C00743 V=800.0 PL=0
MOVL C00744 V=800.0 PL=0
MOVL C00745 V=800.0 PL=0
MOVL C00746 V=800.0 PL=0
MOVL C00747 V=800.0 PL=0
MOVL C00748 V=800.0 PL=0
MOVL C00749 V=800.0 PL=0
MOVL C00750 V=800.0 PL=0
MOVL C00751 V=800.0 PL=0
MOVL C00752 V=800.0 PL=0
MOVL C00753 V=800.0 PL=0
MOVL C00754 V=800.0 PL=0
MOVL C00755 V=800.0 PL=0
MOVL C00756 V=800.0 PL=0
MOVL C00757 V=800.0 PL=0
MOVL C00758 V=800.0 PL=0
MOVL C00759 V=800.0 PL=0
MOVL C00760 V=800.0 PL=0
MOVL C00761 V=800.0 PL=0
MOVL C00762 V=800.0 PL=0
MOVL C00763 V=800.0 PL=0
MOVL C00764 V=800.0 PL=0
MOVL C00765 V=800.0 PL=0
MOVL C00766 V=800.0 PL=0
MOVL C00767 V=800.0 PL=0
MOVL C00768 V=800.0 PL=0
MOVL C00769 V=800.0 PL=0
MOVL C00770 V=800.0 PL=0
MOVL C00771 V=800.0 PL=0
MOVL C00772 V=800.0 PL=0
MOVL C00773 V=800.0 PL=0
MOVL C00774 V=800.0 PL=0
MOVL C00775 V=800.0 PL=0
MOVL C00776 V=800.0 PL=0
MOVL C00777 V=800.0 PL=0
MOVL C00778 V=800.0 PL=0
MOVL C00779 V=800.0 PL=0
MOVL C00780 V=800.0 PL=0
MOVL C00781 V=800.0 PL=0
MOVL C00782 V=800.0 PL=0
MOVL C00783 V=800.0 PL=0
MOVL C00784 V=800.0 PL=0
MOVL C00785 V=800.0 PL=0
MOVL C00786 V=800.0 PL=0
MOVL C00787 V=800.0 PL=0
MOVL C00788 V=800.0 PL=0
MOVL C00789 V=800.0 PL=0
MOVL C00790 V=800.0 PL=0
MOVL C00791 V=800.0 PL=0
MOVL C00792 V=800.0 PL=0
MOVL C00793 V=800.0 PL=0
MOVL C00794 V=800.0 PL=0
MOVL C00795 V=800.0 PL=0
MOVL C00796 V=800.0 PL=0
MOVL C00797 V=800.0 PL=0
MOVL C00798 V=800.0 PL=0
MOVL C00799 V=800.0 PL=0
MOVL C00800 V=800.0 PL=0
MOVL C00801 V=800.0 PL=0
MOVL C00802 V=800.0 PL=0
MOVL C00803 V=800.0 PL=0
MOVL C00804 V=800.0 PL=0
MOVL C00805 V=800.0 PL=0
MOVL C00806 V=800.0 PL=0
MOVL C00807 V=800.0 PL=0
MOVL C00808 V=800.0 PL=0
MOVL C00809 V=800.0 PL=0
MOVL C00810 V=800.0 PL=0
MOVL C00811 V=800.0 PL=0
MOVL C00812 V=800.0 PL=0
MOVL C00813 V=800.0 PL=0
MOVL C00814 V=800.0 PL=0
MOVL C00815 V=800.0 PL=0
MOVL C00816 V=800.0 PL=0
MOVL C00817 V=800.0 PL=0
MOVL C00818 V=800.0 PL=0
MOVL C00819 V=800.0 PL=0
MOVL C00820 V=800.0 PL=0
MOVL C00821 V=800.0 PL=0
MOVL C00822 V=800.0 PL=0
MOVL C00823 V=800.0 PL=0
MOVL C00824 V=800.0 PL=0
MOVL C00825 V=800.0 PL=0
MOVL C00826 V=800.0 PL=0
MOVL C00827 V=800.0 PL=0
MOVL C00828 V=800.0 PL=0
MOVL C00829 V=800.0 PL=0
MOVL C00830 V=800.0 PL=0
MOVL C00831 V=800.0 PL=0
MOVL C00832 V=800.0 PL=0
MOVL C00833 V=800.0 PL=0
MOVL C00834 V=800.0 PL=0
MOVL C00835 V=800.0 PL=0
MOVL C00836 V=800.0 PL=0
MOVL C00837 V=800.0 PL=0
MOVL C00838 V=800.0 PL=0
MOVL C00839 V=800.0 PL=0
MOVL C00840 V=800.0 PL=0
MOVL C00841 V=800.0 PL=0
MOVL C00842 V=800.0 PL=0
MOVL C00843 V=800.0 PL=0
MOVL C00844 V=800.0 PL=0
MOVL C00845 V=800.0 PL=0
MOVL C00846 V=800.0 PL=0
MOVL C00847 V=800.0 PL=0
MOVL C00848 V=800.0 PL=0
MOVL C00849 V=800.0 PL=0
MOVL C00850 V=800.0 PL=0
MOVL C00851 V=800.0 PL=0
MOVL C00852 V=800.0 PL=0
MOVL C00853 V=800.0 PL=0
MOVL C00854 V=800.0 PL=0
MOVL C00855 V=800.0 PL=0
MOVL C00856 V=800.0 PL=0
MOVL C00857 V=800.0 PL=0
MOVL C00858 V=800.0 PL=0
MOVL C00859 V=800.0 PL=0
MOVL C00860 V=800.0 PL=0
MOVL C00861 V=800.0 PL=0
MOVL C00862 V=800.0 PL=0
MOVL C00863 V=800.0 PL=0
MOVL C00864 V=800.0 PL=0
MOVL C00865 V=800.0 PL=0
MOVL C00866 V=800.0 PL=0
MOVL C00867 V=800.0 PL=0
MOVL C00868 V=800.0 PL=0
MOVL C00869 V=800.0 PL=0
MOVL C00870 V=800.0 PL=0
MOVL C00871 V=800.0 PL=0
MOVL C00872 V=800.0 PL=0
MOVL C00873 V=800.0 PL=0
MOVL C00874 V=800.0 PL=0
MOVL C00875 V=800.0 PL=0
MOVL C00876 V=800.0 PL=0
MOVL C00877 V=800.0 PL=0
MOVL C00878 V=800.0 PL=0
MOVL C00879 V=800.0 PL=0
MOVL C00880 V=800.0 PL=0
MOVL C00881 V=800.0 PL=0
MOVL C00882 V=800.0 PL=0
MOVL C00883 V=800.0 PL=0
MOVL C00884 V=800.0 PL=0
MOVL C00885 V=800.0 PL=0
MOVL C00886 V=800.0 PL=0
MOVL C00887 V=800.0 PL=0
MOVL C00888 V=800.0 PL=0
MOVL C00889 V=800.0 PL=0
MOVL C00890 V=800.0 PL=0
MOVL C00891 V=800.0 PL=0
MOVL C00892 V=800.0 PL=0
MOVL C00893 V=800.0 PL=0
MOVL C00894 V=800.0 PL=0
MOVL C00895 V=800.0 PL=0
MOVL C00896 V=800.0 PL=0
MOVL C00897 V=800.0 PL=0
MOVL C00898 V=800.0 PL=0
MOVL C00899 V=800.0 PL=0
MOVL C00900 V=800.0 PL=0
MOVL C00901 V=800.0 PL=0
MOVL C00902 V=800.0 PL=0
MOVL C00903 V=800.0 PL=0
MOVL C00904 V=800.0 PL=0
MOVL C00905 V=800.0 PL=0
MOVL C00906 V=800.0 PL=0
MOVL C00907 V=800.0 PL=0
MOVL C00908 V=800.0 PL=0
MOVL C00909 V=800.0 PL=0
MOVL C00910 V=800.0 PL=0
MOVL C00911 V=800.0 PL=0
MOVL C00912 V=800.0 PL=0
MOVL C00913 V=800.0 PL=0
MOVL C00914 V=800.0 PL=0
MOVL C00915 V=800.0 PL=0
MOVL C00916 V=800.0 PL=0
MOVL C00917 V=800.0 PL=0
MOVL C00918 V=800.0 PL=0
MOVL C00919 V=800.0 PL=0
MOVL C00920 V=800.0 PL=0
MOVL C00921 V=800.0 PL=0
MOVL C00922 V=800.0 PL=0
MOVL C00923 V=800.0 PL=0
MOVL C00924 V=800.0 PL=0
MOVL C00925 V=800.0 PL=0
MOVL C00926 V=800.0 PL=0
MOVL C00927 V=800.0 PL=0
MOVL C00928 V=800.0 PL=0
MOVL C00929 V=800.0 PL=0
MOVL C00930 V=800.0 PL=0
MOVL C00931 V=800.0 PL=0
MOVL C00932 V=800.0 PL=0
MOVL C00933 V=800.0 PL=0
MOVL C00934 V=800.0 PL=0
MOVL C00935 V=800.0 PL=0
MOVL C00936 V=800.0 PL=0
MOVL C00937 V=800.0 PL=0
MOVL C00938 V=800.0 PL=0
MOVL C00939 V=800.0 PL=0
MOVL C00940 V=800.0 PL=0
MOVL C00941 V=800.0 PL=0
MOVL C00942 V=800.0 PL=0
MOVL C00943 V=800.0 PL=0
MOVL C00944 V=800.0 PL=0
MOVL C00945 V=800.0 PL=0
MOVL C00946 V=800.0 PL=0
MOVL C00947 V=800.0 PL=0
MOVL C00948 V=800.0 PL=0
MOVL C00949 V=800.0 PL=0
MOVL C00950 V=800.0 PL=0
MOVL C00951 V=800.0 PL=0
MOVL C00952 V=800.0 PL=0
MOVL C00953 V=800.0 PL=0
MOVL C00954 V=800.0 PL=0
MOVL C00955 V=800.0 PL=0
MOVL C00956 V=800.0 PL=0
MOVL C00957 V=800.0 PL=0
MOVL C00958 V=800.0 PL=0
MOVL C00959 V=800.0 PL=0
MOVL C00960 V=800.0 PL=0
MOVL C00961 V=800.0 PL=0
MOVL C00962 V=800.0 PL=0
MOVL C00963 V=800.0 PL=0
MOVL C00964 V=800.0 PL=0
MOVL C00965 V=800.0 PL=0
MOVL C00966 V=800.0 PL=0
MOVL C00967 V=800.0 PL=0
MOVL C00968 V=800.0 PL=0
MOVL C00969 V=800.0 PL=0
MOVL C00970 V=800.0 PL=0
MOVL C00971 V=800.0 PL=0
MOVL C00972 V=800.0 PL=0
MOVL C00973 V=800.0 PL=0
MOVL C00974 V=800.0 PL=0
MOVL C00975 V=800.0 PL=0
MOVL C00976 V=800.0 PL=0
MOVL C00977 V=800.0 PL=0
MOVL C00978 V=800.0 PL=0
MOVL C00979 V=800.0 PL=0
MOVL C00980 V=800.0 PL=0
MOVL C00981 V=800.0 PL=0
MOVL C00982 V=800.0 PL=0
MOVL C00983 V=800.0 PL=0
MOVL C00984 V=800.0 PL=0
MOVL C00985 V=800.0 PL=0
MOVL C00986 V=800.0 PL=0
MOVL C00987 V=800.0 PL=0
MOVL C00988 V=800.0 PL=0
MOVL C00989 V=800.0 PL=0
MOVL C00990 V=800.0 PL=0
MOVL C00991 V=800.0 PL=0
MOVL C00992 V=800.0 PL=0
MOVL C00993 V=800.0 PL=0
MOVL C00994 V=800.0 PL=0
MOVL C00995 V=800.0 PL=0
MOVL C00996 V=800.0 PL=0
MOVL C00997 V=800.0 PL=0
MOVL C00998 V=800.0 PL=0
MOVL C00999 V=800.0 PL=0
MOVL C01000 V=800.0 PL=0
MOVL C01001 V=800.0 PL=0
MOVL C01002 V=800.0 PL=0
MOVL C01003 V=800.0 PL=0
MOVL C01004 V=800.0 PL=0
MOVL C01005 V=800.0 PL=0
MOVL C01006 V=800.0 PL=0
MOVL C01007 V=800.0 PL=0
MOVL C01008 V=800.0 PL=0
MOVL C01009 V=800.0 PL=0
MOVL C01010 V=800.0 PL=0
MOVL C01011 V=800.0 PL=0
MOVL C01012 V=800.0 PL=0
MOVL C01013 V=800.0 PL=0
MOVL C01014 V=800.0 PL=0
MOVL C01015 V=800.0 PL=0
MOVL C01016 V=800.0 PL=0
MOVL C01017 V=800.0 PL=0
MOVL C01018 V=800.0 PL=0
MOVL C01019 V=800.0 PL=0
MOVL C01020 V=800.0 PL=0
MOVL C01021 V=800.0 PL=0
MOVL C01022 V=800.0 PL=0
MOVL C01023 V=800.0 PL=0
MOVL C01024 V=800.0 PL=0
MOVL C01025 V=800.0 PL=0
MOVL C01026 V=800.0 PL=0
MOVL C01027 V=800.0 PL=0
MOVL C01028 V=800.0 PL=0
MOVL C01029 V=800.0 PL=0
MOVL C01030 V=800.0 PL=0
MOVL C01031 V=800.0 PL=0
MOVL C01032 V=800.0 PL=0
MOVL C01033 V=800.0 PL=0
MOVL C01034 V=800.0 PL=0
MOVL C01035 V=800.0 PL=0
MOVL C01036 V=800.0 PL=0
MOVL C01037 V=800.0 PL=0
MOVL C01038 V=800.0 PL=0
MOVL C01039 V=800.0 PL=0
MOVL C01040 V=800.0 PL=0
MOVL C01041 V=800.0 PL=0
MOVL C01042 V=800.0 PL=0
MOVL C01043 V=800.0 PL=0
MOVL C01044 V=800.0 PL=0
MOVL C01045 V=800.0 PL=0
MOVL C01046 V=800.0 PL=0
MOVL C01047 V=800.0 PL=0
MOVL C01048 V=800.0 PL=0
MOVL C01049 V=800.0 PL=0
MOVL C01050 V=800.0 PL=0
MOVL C01051 V=800.0 PL=0
MOVL C01052 V=800.0 PL=0
MOVL C01053 V=800.0 PL=0
MOVL C01054 V=800.0 PL=0
MOVL C01055 V=800.0 PL=0
MOVL C01056 V=800.0 PL=0
MOVL C01057 V=800.0 PL=0
MOVL C01058 V=800.0 PL=0
MOVL C01059 V=800.0 PL=0
MOVL C01060 V=800.0 PL=0
MOVL C01061 V=800.0 PL=0
MOVL C01062 V=800.0 PL=0
MOVL C01063 V=800.0 PL=0
MOVL C01064 V=800.0 PL=0
MOVL C01065 V=800.0 PL=0
MOVL C01066 V=800.0 PL=0
MOVL C01067 V=800.0 PL=0
MOVL C01068 V=800.0 PL=0
MOVL C01069 V=800.0 PL=0
MOVL C01070 V=800.0 PL=0
MOVL C01071 V=800.0 PL=0
MOVL C01072 V=800.0 PL=0
MOVL C01073 V=800.0 PL=0
MOVL C01074 V=800.0 PL=0
MOVL C01075 V=800.0 PL=0
MOVL C01076 V=800.0 PL=0
MOVL C01077 V=800.0 PL=0
MOVL C01078 V=800.0 PL=0
MOVL C01079 V=800.0 PL=0
MOVL C01080 V=800.0 PL=0
MOVL C01081 V=800.0 PL=0
MOVL C01082 V=800.0 PL=0
MOVL C01083 V=800.0 PL=0
MOVL C01084 V=800.0 PL=0
MOVL C01085 V=800.0 PL=0
MOVL C01086 V=800.0 PL=0
MOVL C01087 V=800.0 PL=0
MOVL C01088 V=800.0 PL=0
MOVL C01089 V=800.0 PL=0
MOVL C01090 V=800.0 PL=0
MOVL C01091 V=800.0 PL=0
MOVL C01092 V=800.0 PL=0
MOVL C01093 V=800.0 PL=0
MOVL C01094 V=800.0 PL=0
MOVL C01095 V=800.0 PL=0
MOVL C01096 V=800.0 PL=0
MOVL C01097 V=800.0 PL=0
MOVL C01098 V=800.0 PL=0
MOVL C01099 V=800.0 PL=0
MOVL C01100 V=800.0 PL=0
MOVL C01101 V=800.0 PL=0
MOVL C01102 V=800.0 PL=0
MOVL C01103 V=800.0 PL=0
MOVL C01104 V=800.0 PL=0
MOVL C01105 V=800.0 PL=0
MOVL C01106 V=800.0 PL=0
MOVL C01107 V=800.0 PL=0
MOVL C01108 V=800.0 PL=0
MOVL C01109 V=800.0 PL=0
MOVL C01110 V=800.0 PL=0
MOVL C01111 V=800.0 PL=0
MOVL C01112 V=800.0 PL=0
MOVL C01113 V=800.0 PL=0
MOVL C01114 V=800.0 PL=0
MOVL C01115 V=800.0 PL=0
MOVL C01116 V=800.0 PL=0
MOVL C01117 V=800.0 PL=0
MOVL C01118 V=800.0 PL=0
MOVL C01119 V=800.0 PL=0
MOVL C01120 V=800.0 PL=0
MOVL C01121 V=800.0 PL=0
MOVL C01122 V=800.0 PL=0
MOVL C01123 V=800.0 PL=0
MOVL C01124 V=800.0 PL=0
MOVL C01125 V=800.0 PL=0
MOVL C01126 V=800.0 PL=0
MOVL C01127 V=800.0 PL=0
MOVL C01128 V=800.0 PL=0
MOVL C01129 V=800.0 PL=0
MOVL C01130 V=800.0 PL=0
MOVL C01131 V=800.0 PL=0
MOVL C01132 V=800.0 PL=0
MOVL C01133 V=800.0 PL=0
MOVL C01134 V=800.0 PL=0
MOVL C01135 V=800.0 PL=0
MOVL C01136 V=800.0 PL=0
MOVL C01137 V=800.0 PL=0
MOVL C01138 V=800.0 PL=0
MOVL C01139 V=800.0 PL=0
MOVL C01140 V=800.0 PL=0
MOVL C01141 V=800.0 PL=0
MOVL C01142 V=800.0 PL=0
MOVL C01143 V=800.0 PL=0
MOVL C01144 V=800.0 PL=0
MOVL C01145 V=800.0 PL=0
MOVL C01146 V=800.0 PL=0
MOVL C01147 V=800.0 PL=0
MOVL C01148 V=800.0 PL=0
MOVL C01149 V=800.0 PL=0
MOVL C01150 V=800.0 PL=0
MOVL C01151 V=800.0 PL=0
MOVL C01152 V=800.0 PL=0
MOVL C01153 V=800.0 PL=0
MOVL C01154 V=800.0 PL=0
MOVL C01155 V=800.0 PL=0
MOVL C01156 V=800.0 PL=0
MOVL C01157 V=800.0 PL=0
MOVL C01158 V=800.0 PL=0
MOVL C01159 V=800.0 PL=0
MOVL C01160 V=800.0 PL=0
MOVL C01161 V=800.0 PL=0
MOVL C01162 V=800.0 PL=0
MOVL C01163 V=800.0 PL=0
MOVL C01164 V=800.0 PL=0
MOVL C01165 V=800.0 PL=0
MOVL C01166 V=800.0 PL=0
MOVL C01167 V=800.0 PL=0
MOVL C01168 V=800.0 PL=0
MOVL C01169 V=800.0 PL=0
MOVL C01170 V=800.0 PL=0
MOVL C01171 V=800.0 PL=0
MOVL C01172 V=800.0 PL=0
MOVL C01173 V=800.0 PL=0
MOVL C01174 V=800.0 PL=0
MOVL C01175 V=800.0 PL=0
MOVL C01176 V=800.0 PL=0
MOVL C01177 V=800.0 PL=0
MOVL C01178 V=800.0 PL=0
MOVL C01179 V=800.0 PL=0
MOVL C01180 V=800.0 PL=0
MOVL C01181 V=800.0 PL=0
MOVL C01182 V=800.0 PL=0
MOVL C01183 V=800.0 PL=0
MOVL C01184 V=800.0 PL=0
MOVL C01185 V=800.0 PL=0
MOVL C01186 V=800.0 PL=0
MOVL C01187 V=800.0 PL=0
MOVL C01188 V=800.0 PL=0
MOVL C01189 V=800.0 PL=0
MOVL C01190 V=800.0 PL=0
MOVL C01191 V=800.0 PL=0
MOVL C01192 V=800.0 PL=0
MOVL C01193 V=800.0 PL=0
MOVL C01194 V=800.0 PL=0
MOVL C01195 V=800.0 PL=0
MOVL C01196 V=800.0 PL=0
MOVL C01197 V=800.0 PL=0
MOVL C01198 V=800.0 PL=0
MOVL C01199 V=800.0 PL=0
MOVL C01200 V=800.0 PL=0
MOVL C01201 V=800.0 PL=0
MOVL C01202 V=800.0 PL=0
MOVL C01203 V=800.0 PL=0
MOVL C01204 V=800.0 PL=0
MOVL C01205 V=800.0 PL=0
MOVL C01206 V=800.0 PL=0
MOVL C01207 V=800.0 PL=0
MOVL C01208 V=800.0 PL=0
MOVL C01209 V=800.0 PL=0
MOVL C01210 V=800.0 PL=0
MOVL C01211 V=800.0 PL=0
MOVL C01212 V=800.0 PL=0
MOVL C01213 V=800.0 PL=0
MOVL C01214 V=800.0 PL=0
MOVL C01215 V=800.0 PL=0
MOVL C01216 V=800.0 PL=0
MOVL C01217 V=800.0 PL=0
MOVL C01218 V=800.0 PL=0
MOVL C01219 V=800.0 PL=0
MOVL C01220 V=800.0 PL=0
MOVL C01221 V=800.0 PL=0
MOVL C01222 V=800.0 PL=0
MOVL C01223 V=800.0 PL=0
MOVL C01224 V=800.0 PL=0
MOVL C01225 V=800.0 PL=0
MOVL C01226 V=800.0 PL=0
MOVL C01227 V=800.0 PL=0
MOVL C01228 V=800.0 PL=0
MOVL C01229 V=800.0 PL=0
MOVL C01230 V=800.0 PL=0
MOVL C01231 V=800.0 PL=0
MOVL C01232 V=800.0 PL=0
MOVL C01233 V=800.0 PL=0
MOVL C01234 V=800.0 PL=0
MOVL C01235 V=800.0 PL=0
MOVL C01236 V=800.0 PL=0
MOVL C01237 V=800.0 PL=0
MOVL C01238 V=800.0 PL=0
MOVL C01239 V=800.0 PL=0
MOVL C01240 V=800.0 PL=0
MOVL C01241 V=800.0 PL=0
MOVL C01242 V=800.0 PL=0
MOVL C01243 V=800.0 PL=0
MOVL C01244 V=800.0 PL=0
MOVL C01245 V=800.0 PL=0
MOVL C01246 V=800.0 PL=0
MOVL C01247 V=800.0 PL=0
MOVL C01248 V=800.0 PL=0
MOVL C01249 V=800.0 PL=0
MOVL C01250 V=800.0 PL=0
MOVL C01251 V=800.0 PL=0
MOVL C01252 V=800.0 PL=0
MOVL C01253 V=800.0 PL=0
MOVL C01254 V=800.0 PL=0
MOVL C01255 V=800.0 PL=0
MOVL C01256 V=800.0 PL=0
MOVL C01257 V=800.0 PL=0
MOVL C01258 V=800.0 PL=0
MOVL C01259 V=800.0 PL=0
MOVL C01260 V=800.0 PL=0
MOVL C01261 V=800.0 PL=0
MOVL C01262 V=800.0 PL=0
MOVL C01263 V=800.0 PL=0
MOVL C01264 V=800.0 PL=0
MOVL C01265 V=800.0 PL=0
MOVL C01266 V=800.0 PL=0
MOVL C01267 V=800.0 PL=0
MOVL C01268 V=800.0 PL=0
MOVL C01269 V=800.0 PL=0
MOVL C01270 V=800.0 PL=0
MOVL C01271 V=800.0 PL=0
MOVL C01272 V=800.0 PL=0
MOVL C01273 V=800.0 PL=0
MOVL C01274 V=800.0 PL=0
MOVL C01275 V=800.0 PL=0
MOVL C01276 V=800.0 PL=0
MOVL C01277 V=800.0 PL=0
MOVL C01278 V=800.0 PL=0
MOVL C01279 V=800.0 PL=0
MOVL C01280 V=800.0 PL=0
MOVL C01281 V=800.0 PL=0
MOVL C01282 V=800.0 PL=0
MOVL C01283 V=800.0 PL=0
MOVL C01284 V=800.0 PL=0
MOVL C01285 V=800.0 PL=0
MOVL C01286 V=800.0 PL=0
MOVL C01287 V=800.0 PL=0
MOVL C01288 V=800.0 PL=0
MOVL C01289 V=800.0 PL=0
MOVL C01290 V=800.0 PL=0
MOVL C01291 V=800.0 PL=0
MOVL C01292 V=800.0 PL=0
MOVL C01293 V=800.0 PL=0
MOVL C01294 V=800.0 PL=0
MOVL C01295 V=800.0 PL=0
MOVL C01296 V=800.0 PL=0
MOVL C01297 V=800.0 PL=0
MOVL C01298 V=800.0 PL=0
MOVL C01299 V=800.0 PL=0
MOVL C01300 V=800.0 PL=0
MOVL C01301 V=800.0 PL=0
MOVL C01302 V=800.0 PL=0
MOVL C01303 V=800.0 PL=0
MOVL C01304 V=800.0 PL=0
MOVL C01305 V=800.0 PL=0
MOVL C01306 V=800.0 PL=0
MOVL C01307 V=800.0 PL=0
MOVL C01308 V=800.0 PL=0
MOVL C01309 V=800.0 PL=0
MOVL C01310 V=800.0 PL=0
MOVL C01311 V=800.0 PL=0
MOVL C01312 V=800.0 PL=0
MOVL C01313 V=800.0 PL=0
MOVL C01314 V=800.0 PL=0
MOVL C01315 V=800.0 PL=0
MOVL C01316 V=800.0 PL=0
MOVL C01317 V=800.0 PL=0
MOVL C01318 V=800.0 PL=0
MOVL C01319 V=800.0 PL=0
MOVL C01320 V=800.0 PL=0
MOVL C01321 V=800.0 PL=0
MOVL C01322 V=800.0 PL=0
MOVL C01323 V=800.0 PL=0
MOVL C01324 V=800.0 PL=0
MOVL C01325 V=800.0 PL=0
MOVL C01326 V=800.0 PL=0
MOVL C01327 V=800.0 PL=0
MOVL C01328 V=800.0 PL=0
MOVL C01329 V=800.0 PL=0
MOVL C01330 V=800.0 PL=0
MOVL C01331 V=800.0 PL=0
MOVL C01332 V=800.0 PL=0
MOVL C01333 V=800.0 PL=0
MOVL C01334 V=800.0 PL=0
MOVL C01335 V=800.0 PL=0
MOVL C01336 V=800.0 PL=0
MOVL C01337 V=800.0 PL=0
MOVL C01338 V=800.0 PL=0
MOVL C01339 V=800.0 PL=0
MOVL C01340 V=800.0 PL=0
MOVL C01341 V=800.0 PL=0
MOVL C01342 V=800.0 PL=0
MOVL C01343 V=800.0 PL=0
MOVL C01344 V=800.0 PL=0
MOVL C01345 V=800.0 PL=0
MOVL C01346 V=800.0 PL=0
MOVL C01347 V=800.0 PL=0
MOVL C01348 V=800.0 PL=0
MOVL C01349 V=800.0 PL=0
MOVL C01350 V=800.0 PL=0
MOVL C01351 V=800.0 PL=0
MOVL C01352 V=800.0 PL=0
MOVL C01353 V=800.0 PL=0
MOVL C01354 V=800.0 PL=0
MOVL C01355 V=800.0 PL=0
MOVL C01356 V=800.0 PL=0
MOVL C01357 V=800.0 PL=0
MOVL C01358 V=800.0 PL=0
MOVL C01359 V=800.0 PL=0
MOVL C01360 V=800.0 PL=0
MOVL C01361 V=800.0 PL=0
MOVL C01362 V=800.0 PL=0
MOVL C01363 V=800.0 PL=0
MOVL C01364 V=800.0 PL=0
MOVL C01365 V=800.0 PL=0
MOVL C01366 V=800.0 PL=0
MOVL C01367 V=800.0 PL=0
MOVL C01368 V=800.0 PL=0
MOVL C01369 V=800.0 PL=0
MOVL C01370 V=800.0 PL=0
MOVL C01371 V=800.0 PL=0
MOVL C01372 V=800.0 PL=0
MOVL C01373 V=800.0 PL=0
MOVL C01374 V=800.0 PL=0
MOVL C01375 V=800.0 PL=0
MOVL C01376 V=800.0 PL=0
MOVL C01377 V=800.0 PL=0
MOVL C01378 V=800.0 PL=0
MOVL C01379 V=800.0 PL=0
MOVL C01380 V=800.0 PL=0
MOVL C01381 V=800.0 PL=0
MOVL C01382 V=800.0 PL=0
MOVL C01383 V=800.0 PL=0
MOVL C01384 V=800.0 PL=0
MOVL C01385 V=800.0 PL=0
MOVL C01386 V=800.0 PL=0
MOVL C01387 V=800.0 PL=0
MOVL C01388 V=800.0 PL=0
MOVL C01389 V=800.0 PL=0
MOVL C01390 V=800.0 PL=0
MOVL C01391 V=800.0 PL=0
MOVL C01392 V=800.0 PL=0
MOVL C01393 V=800.0 PL=0
MOVL C01394 V=800.0 PL=0
MOVL C01395 V=800.0 PL=0
MOVL C01396 V=800.0 PL=0
MOVL C01397 V=800.0 PL=0
MOVL C01398 V=800.0 PL=0
MOVL C01399 V=800.0 PL=0
MOVL C01400 V=800.0 PL=0
MOVL C01401 V=800.0 PL=0
MOVL C01402 V=800.0 PL=0
MOVL C01403 V=800.0 PL=0
MOVL C01404 V=800.0 PL=0
MOVL C01405 V=800.0 PL=0
MOVL C01406 V=800.0 PL=0
MOVL C01407 V=800.0 PL=0
MOVL C01408 V=800.0 PL=0
MOVL C01409 V=800.0 PL=0
MOVL C01410 V=800.0 PL=0
MOVL C01411 V=800.0 PL=0
MOVL C01412 V=800.0 PL=0
MOVL C01413 V=800.0 PL=0
MOVL C01414 V=800.0 PL=0
MOVL C01415 V=800.0 PL=0
MOVL C01416 V=800.0 PL=0
MOVL C01417 V=800.0 PL=0
MOVL C01418 V=800.0 PL=0
MOVL C01419 V=800.0 PL=0
MOVL C01420 V=800.0 PL=0
MOVL C01421 V=800.0 PL=0
MOVL C01422 V=800.0 PL=0
MOVL C01423 V=800.0 PL=0
MOVL C01424 V=800.0 PL=0
MOVL C01425 V=800.0 PL=0
MOVL C01426 V=800.0 PL=0
MOVL C01427 V=800.0 PL=0
MOVL C01428 V=800.0 PL=0
MOVL C01429 V=800.0 PL=0
MOVL C01430 V=800.0 PL=0
MOVL C01431 V=800.0 PL=0
MOVL C01432 V=800.0 PL=0
MOVL C01433 V=800.0 PL=0
MOVL C01434 V=800.0 PL=0
MOVL C01435 V=800.0 PL=0
MOVL C01436 V=800.0 PL=0
MOVL C01437 V=800.0 PL=0
MOVL C01438 V=800.0 PL=0
MOVL C01439 V=800.0 PL=0
MOVL C01440 V=800.0 PL=0
MOVL C01441 V=800.0 PL=0
MOVL C01442 V=800.0 PL=0
MOVL C01443 V=800.0 PL=0
MOVL C01444 V=800.0 PL=0
MOVL C01445 V=800.0 PL=0
MOVL C01446 V=800.0 PL=0
MOVL C01447 V=800.0 PL=0
MOVL C01448 V=800.0 PL=0
MOVL C01449 V=800.0 PL=0
MOVL C01450 V=800.0 PL=0
MOVL C01451 V=800.0 PL=0
MOVL C01452 V=800.0 PL=0
MOVL C01453 V=800.0 PL=0
MOVL C01454 V=800.0 PL=0
MOVL C01455 V=800.0 PL=0
MOVL C01456 V=800.0 PL=0
MOVL C01457 V=800.0 PL=0
MOVL C01458 V=800.0 PL=0
MOVL C01459 V=800.0 PL=0
MOVL C01460 V=800.0 PL=0
MOVL C01461 V=800.0 PL=0
MOVL C01462 V=800.0 PL=0
MOVL C01463 V=800.0 PL=0
MOVL C01464 V=800.0 PL=0
MOVL C01465 V=800.0 PL=0
MOVL C01466 V=800.0 PL=0
MOVL C01467 V=800.0 PL=0
MOVL C01468 V=800.0 PL=0
MOVL C01469 V=800.0 PL=0
MOVL C01470 V=800.0 PL=0
MOVL C01471 V=800.0 PL=0
MOVL C01472 V=800.0 PL=0
MOVL C01473 V=800.0 PL=0
MOVL C01474 V=800.0 PL=0
MOVL C01475 V=800.0 PL=0
MOVL C01476 V=800.0 PL=0
MOVL C01477 V=800.0 PL=0
MOVL C01478 V=800.0 PL=0
MOVL C01479 V=800.0 PL=0
MOVL C01480 V=800.0 PL=0
MOVL C01481 V=800.0 PL=0
MOVL C01482 V=800.0 PL=0
MOVL C01483 V=800.0 PL=0
MOVL C01484 V=800.0 PL=0
MOVL C01485 V=800.0 PL=0
MOVL C01486 V=800.0 PL=0
MOVL C01487 V=800.0 PL=0
MOVL C01488 V=800.0 PL=0
MOVL C01489 V=800.0 PL=0
MOVL C01490 V=800.0 PL=0
MOVL C01491 V=800.0 PL=0
MOVL C01492 V=800.0 PL=0
MOVL C01493 V=800.0 PL=0
MOVL C01494 V=800.0 PL=0
MOVL C01495 V=800.0 PL=0
MOVL C01496 V=800.0 PL=0
MOVL C01497 V=800.0 PL=0
MOVL C01498 V=800.0 PL=0
MOVL C01499 V=800.0 PL=0
MOVL C01500 V=800.0 PL=0
MOVL C01501 V=800.0 PL=0
MOVL C01502 V=800.0 PL=0
MOVL C01503 V=800.0 PL=0
MOVL C01504 V=800.0 PL=0
MOVL C01505 V=800.0 PL=0
MOVL C01506 V=800.0 PL=0
MOVL C01507 V=800.0 PL=0
MOVL C01508 V=800.0 PL=0
MOVL C01509 V=800.0 PL=0
MOVL C01510 V=800.0 PL=0
MOVL C01511 V=800.0 PL=0
MOVL C01512 V=800.0 PL=0
MOVL C01513 V=800.0 PL=0
MOVL C01514 V=800.0 PL=0
MOVL C01515 V=800.0 PL=0
MOVL C01516 V=800.0 PL=0
MOVL C01517 V=800.0 PL=0
MOVL C01518 V=800.0 PL=0
MOVL C01519 V=800.0 PL=0
MOVL C01520 V=800.0 PL=0
MOVL C01521 V=800.0 PL=0
MOVL C01522 V=800.0 PL=0
MOVL C01523 V=800.0 PL=0
MOVL C01524 V=800.0 PL=0
MOVL C01525 V=800.0 PL=0
MOVL C01526 V=800.0 PL=0
MOVL C01527 V=800.0 PL=0
MOVL C01528 V=800.0 PL=0
MOVL C01529 V=800.0 PL=0
MOVL C01530 V=800.0 PL=0
MOVL C01531 V=800.0 PL=0
MOVL C01532 V=800.0 PL=0
MOVL C01533 V=800.0 PL=0
MOVL C01534 V=800.0 PL=0
MOVL C01535 V=800.0 PL=0
MOVL C01536 V=800.0 PL=0
MOVL C01537 V=800.0 PL=0
MOVL C01538 V=800.0 PL=0
MOVL C01539 V=800.0 PL=0
MOVL C01540 V=800.0 PL=0
MOVL C01541 V=800.0 PL=0
MOVL C01542 V=800.0 PL=0
MOVL C01543 V=800.0 PL=0
MOVL C01544 V=800.0 PL=0
MOVL C01545 V=800.0 PL=0
MOVL C01546 V=800.0 PL=0
MOVL C01547 V=800.0 PL=0
MOVL C01548 V=800.0 PL=0
MOVL C01549 V=800.0 PL=0
MOVL C01550 V=800.0 PL=0
MOVL C01551 V=800.0 PL=0
MOVL C01552 V=800.0 PL=0
MOVL C01553 V=800.0 PL=0
MOVL C01554 V=800.0 PL=0
MOVL C01555 V=800.0 PL=0
MOVL C01556 V=800.0 PL=0
MOVL C01557 V=800.0 PL=0
MOVL C01558 V=800.0 PL=0
MOVL C01559 V=800.0 PL=0
MOVL C01560 V=800.0 PL=0
MOVL C01561 V=800.0 PL=0
MOVL C01562 V=800.0 PL=0
MOVL C01563 V=800.0 PL=0
MOVL C01564 V=800.0 PL=0
MOVL C01565 V=800.0 PL=0
MOVL C01566 V=800.0 PL=0
MOVL C01567 V=800.0 PL=0
MOVL C01568 V=800.0 PL=0
MOVL C01569 V=800.0 PL=0
MOVL C01570 V=800.0 PL=0
MOVL C01571 V=800.0 PL=0
MOVL C01572 V=800.0 PL=0
MOVL C01573 V=800.0 PL=0
MOVL C01574 V=800.0 PL=0
MOVL C01575 V=800.0 PL=0
MOVL C01576 V=800.0 PL=0
MOVL C01577 V=800.0 PL=0
MOVL C01578 V=800.0 PL=0
MOVL C01579 V=800.0 PL=0
MOVL C01580 V=800.0 PL=0
MOVL C01581 V=800.0 PL=0
MOVL C01582 V=800.0 PL=0
MOVL C01583 V=800.0 PL=0
MOVL C01584 V=800.0 PL=0
MOVL C01585 V=800.0 PL=0
MOVL C01586 V=800.0 PL=0
MOVL C01587 V=800.0 PL=0
MOVL C01588 V=800.0 PL=0
MOVL C01589 V=800.0 PL=0
MOVL C01590 V=800.0 PL=0
MOVL C01591 V=800.0 PL=0
MOVL C01592 V=800.0 PL=0
MOVL C01593 V=800.0 PL=0
MOVL C01594 V=800.0 PL=0
MOVL C01595 V=800.0 PL=0
MOVL C01596 V=800.0 PL=0
MOVL C01597 V=800.0 PL=0
MOVL C01598 V=800.0 PL=0
MOVL C01599 V=800.0 PL=0
MOVL C01600 V=800.0 PL=0
MOVL C01601 V=800.0 PL=0
MOVL C01602 V=800.0 PL=0
MOVL C01603 V=800.0 PL=0
MOVL C01604 V=800.0 PL=0
MOVL C01605 V=800.0 PL=0
MOVL C01606 V=800.0 PL=0
MOVL C01607 V=800.0 PL=0
MOVL C01608 V=800.0 PL=0
MOVL C01609 V=800.0 PL=0
MOVL C01610 V=800.0 PL=0
MOVL C01611 V=800.0 PL=0
MOVL C01612 V=800.0 PL=0
MOVL C01613 V=800.0 PL=0
MOVL C01614 V=800.0 PL=0
MOVL C01615 V=800.0 PL=0
MOVL C01616 V=800.0 PL=0
MOVL C01617 V=800.0 PL=0
MOVL C01618 V=800.0 PL=0
MOVL C01619 V=800.0 PL=0
MOVL C01620 V=800.0 PL=0
MOVL C01621 V=800.0 PL=0
MOVL C01622 V=800.0 PL=0
MOVL C01623 V=800.0 PL=0
MOVL C01624 V=800.0 PL=0
MOVL C01625 V=800.0 PL=0
MOVL C01626 V=800.0 PL=0
MOVL C01627 V=800.0 PL=0
MOVL C01628 V=800.0 PL=0
MOVL C01629 V=800.0 PL=0
MOVL C01630 V=800.0 PL=0
MOVL C01631 V=800.0 PL=0
MOVL C01632 V=800.0 PL=0
MOVL C01633 V=800.0 PL=0
MOVL C01634 V=800.0 PL=0
MOVL C01635 V=800.0 PL=0
MOVL C01636 V=800.0 PL=0
MOVL C01637 V=800.0 PL=0
MOVL C01638 V=800.0 PL=0
MOVL C01639 V=800.0 PL=0
MOVL C01640 V=800.0 PL=0
MOVL C01641 V=800.0 PL=0
MOVL C01642 V=800.0 PL=0
MOVL C01643 V=800.0 PL=0
MOVL C01644 V=800.0 PL=0
MOVL C01645 V=800.0 PL=0
MOVL C01646 V=800.0 PL=0
MOVL C01647 V=800.0 PL=0
MOVL C01648 V=800.0 PL=0
MOVL C01649 V=800.0 PL=0
MOVL C01650 V=800.0 PL=0
MOVL C01651 V=800.0 PL=0
MOVL C01652 V=800.0 PL=0
MOVL C01653 V=800.0 PL=0
MOVL C01654 V=800.0 PL=0
MOVL C01655 V=800.0 PL=0
MOVL C01656 V=800.0 PL=0
MOVL C01657 V=800.0 PL=0
MOVL C01658 V=800.0 PL=0
MOVL C01659 V=800.0 PL=0
MOVL C01660 V=800.0 PL=0
MOVL C01661 V=800.0 PL=0
MOVL C01662 V=800.0 PL=0
MOVL C01663 V=800.0 PL=0
MOVL C01664 V=800.0 PL=0
MOVL C01665 V=800.0 PL=0
MOVL C01666 V=800.0 PL=0
MOVL C01667 V=800.0 PL=0
MOVL C01668 V=800.0 PL=0
MOVL C01669 V=800.0 PL=0
MOVL C01670 V=800.0 PL=0
MOVL C01671 V=800.0 PL=0
MOVL C01672 V=800.0 PL=0
MOVL C01673 V=800.0 PL=0
MOVL C01674 V=800.0 PL=0
MOVL C01675 V=800.0 PL=0
MOVL C01676 V=800.0 PL=0
MOVL C01677 V=800.0 PL=0
MOVL C01678 V=800.0 PL=0
MOVL C01679 V=800.0 PL=0
MOVL C01680 V=800.0 PL=0
MOVL C01681 V=800.0 PL=0
MOVL C01682 V=800.0 PL=0
MOVL C01683 V=800.0 PL=0
MOVL C01684 V=800.0 PL=0
MOVL C01685 V=800.0 PL=0
MOVL C01686 V=800.0 PL=0
MOVL C01687 V=800.0 PL=0
MOVL C01688 V=800.0 PL=0
MOVL C01689 V=800.0 PL=0
MOVL C01690 V=800.0 PL=0
MOVL C01691 V=800.0 PL=0
MOVL C01692 V=800.0 PL=0
MOVL C01693 V=800.0 PL=0
MOVL C01694 V=800.0 PL=0
MOVL C01695 V=800.0 PL=0
MOVL C01696 V=800.0 PL=0
MOVL C01697 V=800.0 PL=0
MOVL C01698 V=800.0 PL=0
MOVL C01699 V=800.0 PL=0
MOVL C01700 V=800.0 PL=0
MOVL C01701 V=800.0 PL=0
MOVL C01702 V=800.0 PL=0
MOVL C01703 V=800.0 PL=0
MOVL C01704 V=800.0 PL=0
MOVL C01705 V=800.0 PL=0
MOVL C01706 V=800.0 PL=0
MOVL C01707 V=800.0 PL=0
MOVL C01708 V=800.0 PL=0
MOVL C01709 V=800.0 PL=0
MOVL C01710 V=800.0 PL=0
MOVL C01711 V=800.0 PL=0
MOVL C01712 V=800.0 PL=0
MOVL C01713 V=800.0 PL=0
MOVL C01714 V=800.0 PL=0
MOVL C01715 V=800.0 PL=0
MOVL C01716 V=800.0 PL=0
MOVL C01717 V=800.0 PL=0
MOVL C01718 V=800.0 PL=0
MOVL C01719 V=800.0 PL=0
MOVL C01720 V=800.0 PL=0
MOVL C01721 V=800.0 PL=0
MOVL C01722 V=800.0 PL=0
MOVL C01723 V=800.0 PL=0
MOVL C01724 V=800.0 PL=0
MOVL C01725 V=800.0 PL=0
MOVL C01726 V=800.0 PL=0
MOVL C01727 V=800.0 PL=0
MOVL C01728 V=800.0 PL=0
MOVL C01729 V=800.0 PL=0
MOVL C01730 V=800.0 PL=0
MOVL C01731 V=800.0 PL=0
MOVL C01732 V=800.0 PL=0
MOVL C01733 V=800.0 PL=0
MOVL C01734 V=800.0 PL=0
MOVL C01735 V=800.0 PL=0
MOVL C01736 V=800.0 PL=0
MOVL C01737 V=800.0 PL=0
MOVL C01738 V=800.0 PL=0
MOVL C01739 V=800.0 PL=0
MOVL C01740 V=800.0 PL=0
MOVL C01741 V=800.0 PL=0
MOVL C01742 V=800.0 PL=0
MOVL C01743 V=800.0 PL=0
MOVL C01744 V=800.0 PL=0
MOVL C01745 V=800.0 PL=0
MOVL C01746 V=800.0 PL=0
MOVL C01747 V=800.0 PL=0
MOVL C01748 V=800.0 PL=0
MOVL C01749 V=800.0 PL=0
MOVL C01750 V=800.0 PL=0
MOVL C01751 V=800.0 PL=0
MOVL C01752 V=800.0 PL=0
MOVL C01753 V=800.0 PL=0
MOVL C01754 V=800.0 PL=0
MOVL C01755 V=800.0 PL=0
MOVL C01756 V=800.0 PL=0
MOVL C01757 V=800.0 PL=0
MOVL C01758 V=800.0 PL=0
MOVL C01759 V=800.0 PL=0
MOVL C01760 V=800.0 PL=0
MOVL C01761 V=800.0 PL=0
MOVL C01762 V=800.0 PL=0
MOVL C01763 V=800.0 PL=0
MOVL C01764 V=800.0 PL=0
MOVL C01765 V=800.0 PL=0
MOVL C01766 V=800.0 PL=0
MOVL C01767 V=800.0 PL=0
MOVL C01768 V=800.0 PL=0
MOVL C01769 V=800.0 PL=0
MOVL C01770 V=800.0 PL=0
MOVL C01771 V=800.0 PL=0
MOVL C01772 V=800.0 PL=0
MOVL C01773 V=800.0 PL=0
MOVL C01774 V=800.0 PL=0
MOVL C01775 V=800.0 PL=0
MOVL C01776 V=800.0 PL=0
MOVL C01777 V=800.0 PL=0
MOVL C01778 V=800.0 PL=0
MOVL C01779 V=800.0 PL=0
MOVL C01780 V=800.0 PL=0
MOVL C01781 V=800.0 PL=0
MOVL C01782 V=800.0 PL=0
MOVL C01783 V=800.0 PL=0
MOVL C01784 V=800.0 PL=0
MOVL C01785 V=800.0 PL=0
MOVL C01786 V=800.0 PL=0
MOVL C01787 V=800.0 PL=0
MOVL C01788 V=800.0 PL=0
MOVL C01789 V=800.0 PL=0
MOVL C01790 V=800.0 PL=0
MOVL C01791 V=800.0 PL=0
MOVL C01792 V=800.0 PL=0
MOVL C01793 V=800.0 PL=0
MOVL C01794 V=800.0 PL=0
MOVL C01795 V=800.0 PL=0
MOVL C01796 V=800.0 PL=0
MOVL C01797 V=800.0 PL=0
MOVL C01798 V=800.0 PL=0
MOVL C01799 V=800.0 PL=0
MOVL C01800 V=800.0 PL=0
MOVL C01801 V=800.0 PL=0
MOVL C01802 V=800.0 PL=0
MOVL C01803 V=800.0 PL=0
MOVL C01804 V=800.0 PL=0
MOVL C01805 V=800.0 PL=0
MOVL C01806 V=800.0 PL=0
MOVL C01807 V=800.0 PL=0
MOVL C01808 V=800.0 PL=0
MOVL C01809 V=800.0 PL=0
MOVL C01810 V=800.0 PL=0
MOVL C01811 V=800.0 PL=0
MOVL C01812 V=800.0 PL=0
MOVL C01813 V=800.0 PL=0
MOVL C01814 V=800.0 PL=0
MOVL C01815 V=800.0 PL=0
MOVL C01816 V=800.0 PL=0
MOVL C01817 V=800.0 PL=0
MOVL C01818 V=800.0 PL=0
MOVL C01819 V=800.0 PL=0
MOVL C01820 V=800.0 PL=0
MOVL C01821 V=800.0 PL=0
MOVL C01822 V=800.0 PL=0
MOVL C01823 V=800.0 PL=0
MOVL C01824 V=800.0 PL=0
MOVL C01825 V=800.0 PL=0
MOVL C01826 V=800.0 PL=0
MOVL C01827 V=800.0 PL=0
MOVL C01828 V=800.0 PL=0
MOVL C01829 V=800.0 PL=0
MOVL C01830 V=800.0 PL=0
MOVL C01831 V=800.0 PL=0
MOVL C01832 V=800.0 PL=0
MOVL C01833 V=800.0 PL=0
MOVL C01834 V=800.0 PL=0
MOVL C01835 V=800.0 PL=0
MOVL C01836 V=800.0 PL=0
MOVL C01837 V=800.0 PL=0
MOVL C01838 V=800.0 PL=0
MOVL C01839 V=800.0 PL=0
MOVL C01840 V=800.0 PL=0
MOVL C01841 V=800.0 PL=0
MOVL C01842 V=800.0 PL=0
MOVL C01843 V=800.0 PL=0
MOVL C01844 V=800.0 PL=0
MOVL C01845 V=800.0 PL=0
MOVL C01846 V=800.0 PL=0
MOVL C01847 V=800.0 PL=0
MOVL C01848 V=800.0 PL=0
MOVL C01849 V=800.0 PL=0
MOVL C01850 V=800.0 PL=0
MOVL C01851 V=800.0 PL=0
MOVL C01852 V=800.0 PL=0
MOVL C01853 V=800.0 PL=0
MOVL C01854 V=800.0 PL=0
MOVL C01855 V=800.0 PL=0
MOVL C01856 V=800.0 PL=0
MOVL C01857 V=800.0 PL=0
MOVL C01858 V=800.0 PL=0
MOVL C01859 V=800.0 PL=0
MOVL C01860 V=800.0 PL=0
MOVL C01861 V=800.0 PL=0
MOVL C01862 V=800.0 PL=0
MOVL C01863 V=800.0 PL=0
MOVL C01864 V=800.0 PL=0
MOVL C01865 V=800.0 PL=0
MOVL C01866 V=800.0 PL=0
MOVL C01867 V=800.0 PL=0
MOVL C01868 V=800.0 PL=0
MOVL C01869 V=800.0 PL=0
MOVL C01870 V=800.0 PL=0
MOVL C01871 V=800.0 PL=0
MOVL C01872 V=800.0 PL=0
MOVL C01873 V=800.0 PL=0
MOVL C01874 V=800.0 PL=0
MOVL C01875 V=800.0 PL=0
MOVL C01876 V=800.0 PL=0
MOVL C01877 V=800.0 PL=0
MOVL C01878 V=800.0 PL=0
MOVL C01879 V=800.0 PL=0
MOVL C01880 V=800.0 PL=0
MOVL C01881 V=800.0 PL=0
MOVL C01882 V=800.0 PL=0
MOVL C01883 V=800.0 PL=0
MOVL C01884 V=800.0 PL=0
MOVL C01885 V=800.0 PL=0
MOVL C01886 V=800.0 PL=0
MOVL C01887 V=800.0 PL=0
MOVL C01888 V=800.0 PL=0
MOVL C01889 V=800.0 PL=0
MOVL C01890 V=800.0 PL=0
MOVL C01891 V=800.0 PL=0
MOVL C01892 V=800.0 PL=0
MOVL C01893 V=800.0 PL=0
MOVL C01894 V=800.0 PL=0
MOVL C01895 V=800.0 PL=0
MOVL C01896 V=800.0 PL=0
MOVL C01897 V=800.0 PL=0
MOVL C01898 V=800.0 PL=0
MOVL C01899 V=800.0 PL=0
MOVL C01900 V=800.0 PL=0
MOVL C01901 V=800.0 PL=0
MOVL C01902 V=800.0 PL=0
MOVL C01903 V=800.0 PL=0
MOVL C01904 V=800.0 PL=0
MOVL C01905 V=800.0 PL=0
MOVL C01906 V=800.0 PL=0
MOVL C01907 V=800.0 PL=0
MOVL C01908 V=800.0 PL=0
MOVL C01909 V=800.0 PL=0
MOVL C01910 V=800.0 PL=0
MOVL C01911 V=800.0 PL=0
MOVL C01912 V=800.0 PL=0
MOVL C01913 V=800.0 PL=0
MOVL C01914 V=800.0 PL=0
MOVL C01915 V=800.0 PL=0
MOVL C01916 V=800.0 PL=0
MOVL C01917 V=800.0 PL=0
MOVL C01918 V=800.0 PL=0
MOVL C01919 V=800.0 PL=0
MOVL C01920 V=800.0 PL=0
MOVL C01921 V=800.0 PL=0
MOVL C01922 V=800.0 PL=0
MOVL C01923 V=800.0 PL=0
MOVL C01924 V=800.0 PL=0
MOVL C01925 V=800.0 PL=0
MOVL C01926 V=800.0 PL=0
MOVL C01927 V=800.0 PL=0
MOVL C01928 V=800.0 PL=0
MOVL C01929 V=800.0 PL=0
MOVL C01930 V=800.0 PL=0
MOVL C01931 V=800.0 PL=0
MOVL C01932 V=800.0 PL=0
MOVL C01933 V=800.0 PL=0
MOVL C01934 V=800.0 PL=0
MOVL C01935 V=800.0 PL=0
MOVL C01936 V=800.0 PL=0
MOVL C01937 V=800.0 PL=0
MOVL C01938 V=800.0 PL=0
MOVL C01939 V=800.0 PL=0
MOVL C01940 V=800.0 PL=0
MOVL C01941 V=800.0 PL=0
MOVL C01942 V=800.0 PL=0
MOVL C01943 V=800.0 PL=0
MOVL C01944 V=800.0 PL=0
MOVL C01945 V=800.0 PL=0
MOVL C01946 V=800.0 PL=0
MOVL C01947 V=800.0 PL=0
MOVL C01948 V=800.0 PL=0
MOVL C01949 V=800.0 PL=0
MOVL C01950 V=800.0 PL=0
MOVL C01951 V=800.0 PL=0
MOVL C01952 V=800.0 PL=0
MOVL C01953 V=800.0 PL=0
MOVL C01954 V=800.0 PL=0
MOVL C01955 V=800.0 PL=0
MOVL C01956 V=800.0 PL=0
MOVL C01957 V=800.0 PL=0
MOVL C01958 V=800.0 PL=0
MOVL C01959 V=800.0 PL=0
MOVL C01960 V=800.0 PL=0
MOVL C01961 V=800.0 PL=0
MOVL C01962 V=800.0 PL=0
MOVL C01963 V=800.0 PL=0
MOVL C01964 V=800.0 PL=0
MOVL C01965 V=800.0 PL=0
MOVL C01966 V=800.0 PL=0
MOVL C01967 V=800.0 PL=0
MOVL C01968 V=800.0 PL=0
MOVL C01969 V=800.0 PL=0
MOVL C01970 V=800.0 PL=0
MOVL C01971 V=800.0 PL=0
MOVL C01972 V=800.0 PL=0
MOVL C01973 V=800.0 PL=0
MOVL C01974 V=800.0 PL=0
MOVL C01975 V=800.0 PL=0
MOVL C01976 V=800.0 PL=0
MOVL C01977 V=800.0 PL=0
MOVL C01978 V=800.0 PL=0
MOVL C01979 V=800.0 PL=0
MOVL C01980 V=800.0 PL=0
MOVL C01981 V=800.0 PL=0
MOVL C01982 V=800.0 PL=0
MOVL C01983 V=800.0 PL=0
MOVL C01984 V=800.0 PL=0
MOVL C01985 V=800.0 PL=0
MOVL C01986 V=800.0 PL=0
MOVL C01987 V=800.0 PL=0
MOVL C01988 V=800.0 PL=0
MOVL C01989 V=800.0 PL=0
MOVL C01990 V=800.0 PL=0
MOVL C01991 V=800.0 PL=0
MOVL C01992 V=800.0 PL=0
MOVL C01993 V=800.0 PL=0
MOVL C01994 V=800.0 PL=0
MOVL C01995 V=800.0 PL=0
MOVL C01996 V=800.0 PL=0
MOVL C01997 V=800.0 PL=0
MOVL C01998 V=800.0 PL=0
MOVL C01999 V=800.0 PL=0
MOVL C02000 V=800.0 PL=0
MOVL C02001 V=800.0 PL=0
MOVL C02002 V=800.0 PL=0
MOVL C02003 V=800.0 PL=0
MOVL C02004 V=800.0 PL=0
MOVL C02005 V=800.0 PL=0
MOVL C02006 V=800.0 PL=0
MOVL C02007 V=800.0 PL=0
MOVL C02008 V=800.0 PL=0
MOVL C02009 V=800.0 PL=0
MOVL C02010 V=800.0 PL=0
MOVL C02011 V=800.0 PL=0
MOVL C02012 V=800.0 PL=0
MOVL C02013 V=800.0 PL=0
MOVL C02014 V=800.0 PL=0
MOVL C02015 V=800.0 PL=0
MOVL C02016 V=800.0 PL=0
MOVL C02017 V=800.0 PL=0
MOVL C02018 V=800.0 PL=0
MOVL C02019 V=800.0 PL=0
MOVL C02020 V=800.0 PL=0
MOVL C02021 V=800.0 PL=0
MOVL C02022 V=800.0 PL=0
MOVL C02023 V=800.0 PL=0
MOVL C02024 V=800.0 PL=0
MOVL C02025 V=800.0 PL=0
MOVL C02026 V=800.0 PL=0
MOVL C02027 V=800.0 PL=0
MOVL C02028 V=800.0 PL=0
MOVL C02029 V=800.0 PL=0
MOVL C02030 V=800.0 PL=0
MOVL C02031 V=800.0 PL=0
MOVL C02032 V=800.0 PL=0
MOVL C02033 V=800.0 PL=0
MOVL C02034 V=800.0 PL=0
MOVL C02035 V=800.0 PL=0
MOVL C02036 V=800.0 PL=0
MOVL C02037 V=800.0 PL=0
MOVL C02038 V=800.0 PL=0
MOVL C02039 V=800.0 PL=0
MOVL C02040 V=800.0 PL=0
MOVL C02041 V=800.0 PL=0
MOVL C02042 V=800.0 PL=0
MOVL C02043 V=800.0 PL=0
MOVL C02044 V=800.0 PL=0
MOVL C02045 V=800.0 PL=0
MOVL C02046 V=800.0 PL=0
MOVL C02047 V=800.0 PL=0
MOVL C02048 V=800.0 PL=0
MOVL C02049 V=800.0 PL=0
MOVL C02050 V=800.0 PL=0
MOVL C02051 V=800.0 PL=0
MOVL C02052 V=800.0 PL=0
MOVL C02053 V=800.0 PL=0
MOVL C02054 V=800.0 PL=0
MOVL C02055 V=800.0 PL=0
MOVL C02056 V=800.0 PL=0
MOVL C02057 V=800.0 PL=0
MOVL C02058 V=800.0 PL=0
MOVL C02059 V=800.0 PL=0
MOVL C02060 V=800.0 PL=0
MOVL C02061 V=800.0 PL=0
MOVL C02062 V=800.0 PL=0
MOVL C02063 V=800.0 PL=0
MOVL C02064 V=800.0 PL=0
MOVL C02065 V=800.0 PL=0
MOVL C02066 V=800.0 PL=0
MOVL C02067 V=800.0 PL=0
MOVL C02068 V=800.0 PL=0
MOVL C02069 V=800.0 PL=0
MOVL C02070 V=800.0 PL=0
MOVL C02071 V=800.0 PL=0
MOVL C02072 V=800.0 PL=0
MOVL C02073 V=800.0 PL=0
MOVL C02074 V=800.0 PL=0
MOVL C02075 V=800.0 PL=0
MOVL C02076 V=800.0 PL=0
MOVL C02077 V=800.0 PL=0
MOVL C02078 V=800.0 PL=0
MOVL C02079 V=800.0 PL=0
MOVL C02080 V=800.0 PL=0
MOVL C02081 V=800.0 PL=0
MOVL C02082 V=800.0 PL=0
MOVL C02083 V=800.0 PL=0
MOVL C02084 V=800.0 PL=0
MOVL C02085 V=800.0 PL=0
MOVL C02086 V=800.0 PL=0
MOVL C02087 V=800.0 PL=0
MOVL C02088 V=800.0 PL=0
MOVL C02089 V=800.0 PL=0
MOVL C02090 V=800.0 PL=0
MOVL C02091 V=800.0 PL=0
MOVL C02092 V=800.0 PL=0
MOVL C02093 V=800.0 PL=0
MOVL C02094 V=800.0 PL=0
MOVL C02095 V=800.0 PL=0
MOVL C02096 V=800.0 PL=0
MOVL C02097 V=800.0 PL=0
MOVL C02098 V=800.0 PL=0
MOVL C02099 V=800.0 PL=0
MOVL C02100 V=800.0 PL=0
MOVL C02101 V=800.0 PL=0
MOVL C02102 V=800.0 PL=0
MOVL C02103 V=800.0 PL=0
MOVL C02104 V=800.0 PL=0
MOVL C02105 V=800.0 PL=0
MOVL C02106 V=800.0 PL=0
MOVL C02107 V=800.0 PL=0
MOVL C02108 V=800.0 PL=0
MOVL C02109 V=800.0 PL=0
MOVL C02110 V=800.0 PL=0
MOVL C02111 V=800.0 PL=0
MOVL C02112 V=800.0 PL=0
MOVL C02113 V=800.0 PL=0
MOVL C02114 V=800.0 PL=0
MOVL C02115 V=800.0 PL=0
MOVL C02116 V=800.0 PL=0
MOVL C02117 V=800.0 PL=0
MOVL C02118 V=800.0 PL=0
MOVL C02119 V=800.0 PL=0
